C08996=1031.211,97.097,-98.859,168.789,43.801,158.206
C08997=1031.206,96.848,-98.839,168.786,43.803,158.206
C08998=1031.199,96.599,-98.821,168.784,43.804,158.206
C08999=1031.194,96.349,-98.802,168.781,43.806,158.206
C09000=1031.187,96.101,-98.782,168.779,43.808,158.206
C09001=1031.180,95.852,-98.764,168.776,43.809,158.206
C09002=1031.175,95.602,-98.744,168.775,43.811,158.206
C09003=1031.168,95.353,-98.726,168.772,43.812,158.206
C09004=1031.163,95.104,-98.706,168.769,43.814,158.207
C09005=1031.156,94.855,-98.688,168.768,43.816,158.207
C09006=1031.150,94.605,-98.669,168.765,43.818,158.207
C09007=1031.144,94.356,-98.650,168.762,43.819,158.207
C09008=1031.138,94.107,-98.631,168.760,43.821,158.207
C09009=1031.132,93.858,-98.612,168.758,43.823,158.207
C09010=1031.125,93.609,-98.593,168.755,43.824,158.207
C09011=1031.120,93.360,-98.573,168.753,43.826,158.207
C09012=1031.113,93.111,-98.555,168.751,43.827,158.208
C09013=1031.107,92.861,-98.535,168.748,43.829,158.208
C09014=1031.101,92.576,-98.514,168.746,43.831,158.208
C09015=1031.093,92.290,-98.492,168.743,43.833,158.208
C09016=1031.086,92.005,-98.470,168.741,43.835,158.208
C09017=1031.079,91.720,-98.449,168.737,43.836,158.208
C09018=1031.073,91.470,-98.431,168.735,43.838,158.208
C09019=1031.067,91.221,-98.411,168.733,43.840,158.208
C09020=1031.061,90.972,-98.393,168.730,43.842,158.209
C09021=1031.055,90.722,-98.373,168.728,43.843,158.209
C09022=1031.049,90.473,-98.355,168.726,43.845,158.209
C09023=1031.043,90.224,-98.336,168.723,43.847,158.209
C09024=1031.037,89.975,-98.317,168.721,43.848,158.209
C09025=1031.031,89.725,-98.298,168.718,43.850,158.209
C09026=1031.024,89.476,-98.279,168.716,43.851,158.209
C09027=1031.018,89.227,-98.260,168.713,43.853,158.209
C09028=1031.012,88.978,-98.242,168.712,43.855,158.210
C09029=1031.005,88.728,-98.224,168.709,43.856,158.210
C09030=1031.000,88.480,-98.206,168.706,43.858,158.210
C09031=1030.993,88.231,-98.187,168.704,43.860,158.210
C09032=1030.988,87.981,-98.168,168.702,43.862,158.210
C09033=1030.981,87.732,-98.149,168.699,43.864,158.210
C09034=1030.975,87.483,-98.130,168.697,43.865,158.210
C09035=1030.969,87.233,-98.112,168.695,43.866,158.210
C09036=1030.962,86.984,-98.094,168.692,43.868,158.210
C09037=1030.956,86.735,-98.075,168.690,43.870,158.211
C09038=1030.949,86.486,-98.056,168.687,43.872,158.211
C09039=1030.943,86.236,-98.038,168.686,43.874,158.211
C09040=1030.937,85.987,-98.019,168.683,43.876,158.211
C09041=1030.931,85.738,-98.001,168.680,43.877,158.211
C09042=1030.925,85.489,-97.982,168.678,43.879,158.211
C09043=1030.919,85.240,-97.964,168.676,43.881,158.211
C09044=1030.913,84.990,-97.946,168.673,43.882,158.211
C09045=1030.906,84.741,-97.927,168.671,43.884,158.212
C09046=1030.900,84.492,-97.908,168.669,43.885,158.212
C09047=1030.894,84.242,-97.890,168.666,43.887,158.212
C09048=1030.888,83.993,-97.871,168.664,43.889,158.212
C09049=1030.882,83.744,-97.853,168.661,43.891,158.212
C09050=1030.876,83.495,-97.834,168.659,43.892,158.212
C09051=1030.870,83.246,-97.816,168.657,43.894,158.212
C09052=1030.863,82.997,-97.798,168.654,43.896,158.212
C09053=1030.857,82.747,-97.779,168.653,43.898,158.213
C09054=1030.851,82.498,-97.761,168.650,43.899,158.213
C09055=1030.844,82.249,-97.743,168.647,43.901,158.213
C09056=1030.839,81.999,-97.723,168.646,43.902,158.213
C09057=1030.833,81.750,-97.706,168.643,43.904,158.213
C09058=1030.827,81.501,-97.687,168.640,43.906,158.213
C09059=1030.820,81.252,-97.668,168.637,43.907,158.213
C09060=1030.814,81.002,-97.650,168.636,43.909,158.213
C09061=1030.808,80.753,-97.632,168.633,43.911,158.213
C09062=1030.802,80.505,-97.614,168.631,43.913,158.214
C09063=1030.796,80.255,-97.596,168.629,43.914,158.214
C09064=1030.789,80.006,-97.577,168.626,43.916,158.214
C09065=1030.784,79.756,-97.558,168.624,43.918,158.214
C09066=1030.777,79.506,-97.540,168.622,43.919,158.214
C09067=1030.772,79.258,-97.522,168.619,43.921,158.214
C09068=1030.766,79.008,-97.504,168.617,43.923,158.214
C09069=1030.759,78.759,-97.485,168.615,43.924,158.214
C09070=1030.753,78.509,-97.467,168.612,43.926,158.215
C09071=1030.747,78.261,-97.449,168.610,43.927,158.215
C09072=1030.741,78.011,-97.431,168.608,43.929,158.215
C09073=1030.735,77.762,-97.412,168.605,43.931,158.215
C09074=1030.728,77.512,-97.394,168.603,43.933,158.215
C09075=1030.722,77.263,-97.376,168.600,43.934,158.215
C09076=1030.717,77.014,-97.358,168.598,43.936,158.215
C09077=1030.710,76.765,-97.339,168.596,43.938,158.215
C09078=1030.703,76.480,-97.319,168.593,43.940,158.215
C09079=1030.696,76.195,-97.298,168.591,43.941,158.216
C09080=1030.689,75.908,-97.277,168.588,43.943,158.216
C09081=1030.682,75.623,-97.257,168.585,43.946,158.216
C09082=1030.676,75.374,-97.238,168.583,43.947,158.216
C09083=1030.669,75.124,-97.221,168.580,43.949,158.216
C09084=1030.663,74.876,-97.203,168.578,43.951,158.216
C09085=1030.657,74.626,-97.185,168.576,43.953,158.216
C09086=1030.651,74.377,-97.167,168.573,43.955,158.217
C09087=1030.644,74.127,-97.148,168.571,43.956,158.217
C09088=1030.639,73.878,-97.130,168.568,43.958,158.217
C09089=1030.632,73.629,-97.113,168.566,43.959,158.217
C09090=1030.625,73.380,-97.094,168.564,43.961,158.217
C09091=1030.620,73.131,-97.077,168.561,43.963,158.217
C09092=1030.614,72.881,-97.059,168.560,43.965,158.217
C09093=1030.607,72.632,-97.040,168.557,43.967,158.218
C09094=1030.601,72.382,-97.022,168.554,43.968,158.218
C09095=1030.595,72.133,-97.005,168.552,43.970,158.218
C09096=1030.589,71.884,-96.987,168.550,43.972,158.218
C09097=1030.582,71.635,-96.969,168.547,43.973,158.218
C09098=1030.577,71.386,-96.951,168.545,43.975,158.218
C09099=1030.571,71.136,-96.933,168.543,43.976,158.218
C09100=1030.564,70.887,-96.915,168.540,43.978,158.218
C09101=1030.558,70.638,-96.898,168.538,43.980,158.218
C09102=1030.552,70.388,-96.880,168.536,43.982,158.219
C09103=1030.546,70.139,-96.861,168.534,43.984,158.219
C09104=1030.539,69.890,-96.844,168.531,43.985,158.219
C09105=1030.533,69.641,-96.826,168.528,43.987,158.219
C09106=1030.527,69.391,-96.808,168.526,43.989,158.219
C09107=1030.522,69.142,-96.791,168.524,43.991,158.219
C09108=1030.515,68.893,-96.772,168.521,43.992,158.219
C09109=1030.508,68.643,-96.755,168.520,43.994,158.219
C09110=1030.503,68.394,-96.737,168.517,43.995,158.219
C09111=1030.496,68.145,-96.720,168.514,43.997,158.220
C09112=1030.490,67.895,-96.702,168.512,43.999,158.220
C09113=1030.484,67.646,-96.684,168.510,44.001,158.220
C09114=1030.477,67.397,-96.666,168.507,44.003,158.220
C09115=1030.471,67.147,-96.648,168.505,44.005,158.220
C09116=1030.466,66.898,-96.631,168.503,44.006,158.220
C09117=1030.459,66.649,-96.613,168.500,44.008,158.220
C09118=1030.453,66.399,-96.595,168.498,44.010,158.221
C09119=1030.447,66.150,-96.578,168.495,44.011,158.221
C09120=1030.440,65.901,-96.561,168.494,44.013,158.221
C09121=1030.435,65.652,-96.543,168.491,44.015,158.221
C09122=1030.428,65.402,-96.526,168.488,44.017,158.221
C09123=1030.422,65.153,-96.508,168.487,44.019,158.221
C09124=1030.416,64.904,-96.490,168.484,44.020,158.221
C09125=1030.409,64.654,-96.473,168.481,44.022,158.221
C09126=1030.403,64.406,-96.455,168.479,44.024,158.222
C09127=1030.397,64.156,-96.437,168.477,44.025,158.222
C09128=1030.390,63.907,-96.419,168.475,44.027,158.222
C09129=1030.384,63.658,-96.402,168.472,44.029,158.222
C09130=1030.378,63.408,-96.384,168.469,44.030,158.222
C09131=1030.372,63.159,-96.368,168.468,44.032,158.222
C09132=1030.366,62.909,-96.350,168.465,44.034,158.222
C09133=1030.359,62.660,-96.333,168.463,44.037,158.223
C09134=1030.353,62.411,-96.316,168.460,44.039,158.223
C09135=1030.346,62.161,-96.299,168.458,44.040,158.223
C09136=1030.341,61.912,-96.281,168.456,44.042,158.223
C09137=1030.334,61.663,-96.264,168.453,44.043,158.223
C09138=1030.327,61.413,-96.246,168.450,44.045,158.223
C09139=1030.321,61.164,-96.229,168.449,44.047,158.223
C09140=1030.315,60.914,-96.212,168.446,44.049,158.223
C09141=1030.308,60.666,-96.195,168.444,44.051,158.224
C09142=1030.302,60.380,-96.175,168.441,44.053,158.224
C09143=1030.294,60.095,-96.155,168.439,44.055,158.224
C09144=1030.287,59.809,-96.135,168.435,44.057,158.224
C09145=1030.280,59.523,-96.115,168.432,44.059,158.224
C09146=1030.273,59.274,-96.098,168.431,44.061,158.224
C09147=1030.267,59.024,-96.082,168.428,44.063,158.224
C09148=1030.260,58.775,-96.064,168.426,44.065,158.225
C09149=1030.254,58.526,-96.047,168.423,44.067,158.225
C09150=1030.248,58.276,-96.029,168.421,44.068,158.225
C09151=1030.241,58.027,-96.012,168.419,44.070,158.225
C09152=1030.235,57.777,-95.995,168.416,44.072,158.225
C09153=1030.229,57.528,-95.978,168.414,44.074,158.225
C09154=1030.222,57.279,-95.961,168.412,44.076,158.226
C09155=1030.216,57.030,-95.944,168.409,44.078,158.226
C09156=1030.210,56.780,-95.927,168.407,44.080,158.226
C09157=1030.204,56.531,-95.910,168.404,44.082,158.226
C09158=1030.197,56.282,-95.892,168.402,44.084,158.226
C09159=1030.191,56.033,-95.875,168.400,44.085,158.226
C09160=1030.185,55.783,-95.858,168.397,44.087,158.226
C09161=1030.179,55.534,-95.841,168.395,44.088,158.226
C09162=1030.172,55.284,-95.824,168.393,44.090,158.227
C09163=1030.167,55.035,-95.807,168.390,44.092,158.227
C09164=1030.160,54.785,-95.790,168.388,44.094,158.227
C09165=1030.154,54.537,-95.773,168.385,44.096,158.227
C09166=1030.147,54.287,-95.756,168.384,44.098,158.227
C09167=1030.142,54.038,-95.739,168.381,44.100,158.227
C09168=1030.135,53.789,-95.722,168.378,44.101,158.227
C09169=1030.129,53.539,-95.705,168.376,44.103,158.227
C09170=1030.123,53.290,-95.688,168.374,44.105,158.228
C09171=1030.116,53.040,-95.670,168.371,44.106,158.228
C09172=1030.110,52.791,-95.654,168.369,44.108,158.228
C09173=1030.104,52.542,-95.636,168.366,44.110,158.228
C09174=1030.097,52.293,-95.619,168.365,44.112,158.228
C09175=1030.092,52.043,-95.603,168.362,44.114,158.228
C09176=1030.085,51.794,-95.585,168.359,44.116,158.228
C09177=1030.079,51.544,-95.569,168.357,44.118,158.228
C09178=1030.072,51.295,-95.552,168.355,44.119,158.229
C09179=1030.067,51.046,-95.534,168.352,44.121,158.229
C09180=1030.060,50.796,-95.517,168.350,44.122,158.229
C09181=1030.054,50.547,-95.501,168.347,44.124,158.229
C09182=1030.048,50.298,-95.484,168.346,44.126,158.229
C09183=1030.042,50.048,-95.466,168.343,44.128,158.229
C09184=1030.036,49.799,-95.450,168.340,44.130,158.229
C09185=1030.030,49.550,-95.433,168.339,44.131,158.229
C09186=1030.023,49.300,-95.416,168.336,44.133,158.230
C09187=1030.018,49.051,-95.399,168.333,44.135,158.230
C09188=1030.011,48.801,-95.382,168.331,44.137,158.230
C09189=1030.005,48.552,-95.365,168.329,44.138,158.230
C09190=1029.999,48.303,-95.349,168.326,44.140,158.230
C09191=1029.993,48.053,-95.331,168.324,44.142,158.230
C09192=1029.987,47.804,-95.315,168.322,44.143,158.230
C09193=1029.981,47.555,-95.298,168.320,44.145,158.230
C09194=1029.974,47.305,-95.281,168.317,44.147,158.230
C09195=1029.969,47.056,-95.264,168.314,44.149,158.231
C09196=1029.963,46.806,-95.247,168.313,44.150,158.231
C09197=1029.956,46.557,-95.230,168.310,44.152,158.231
C09198=1029.950,46.308,-95.214,168.307,44.154,158.231
C09199=1029.944,46.059,-95.196,168.305,44.156,158.231
C09200=1029.938,45.809,-95.180,168.303,44.157,158.231
C09201=1029.932,45.560,-95.163,168.300,44.159,158.231
C09202=1029.926,45.311,-95.146,168.298,44.161,158.231
C09203=1029.919,45.062,-95.129,168.296,44.162,158.232
C09204=1029.913,44.811,-95.112,168.294,44.164,158.232
C09205=1029.908,44.562,-95.096,168.291,44.166,158.232
C09206=1029.900,44.276,-95.077,168.288,44.168,158.232
C09207=1029.894,43.991,-95.058,168.286,44.169,158.232
C09208=1029.887,43.705,-95.038,168.283,44.171,158.232
C09209=1029.879,43.418,-95.019,168.280,44.173,158.232
C09210=1029.873,43.170,-95.002,168.278,44.175,158.232
C09211=1029.868,42.920,-94.985,168.275,44.177,158.232
C09212=1029.861,42.670,-94.969,168.274,44.179,158.233
C09213=1029.855,42.421,-94.953,168.271,44.181,158.233
C09214=1029.848,42.172,-94.936,168.268,44.183,158.233
C09215=1029.843,41.923,-94.920,168.266,44.185,158.233
C09216=1029.836,41.673,-94.903,168.264,44.186,158.233
C09217=1029.830,41.423,-94.887,168.261,44.188,158.233
C09218=1029.824,41.175,-94.870,168.259,44.189,158.233
C09219=1029.817,40.925,-94.853,168.256,44.191,158.233
C09220=1029.811,40.675,-94.837,168.254,44.193,158.233
C09221=1029.805,40.426,-94.821,168.252,44.195,158.234
C09222=1029.799,40.177,-94.804,168.249,44.197,158.234
C09223=1029.792,39.927,-94.787,168.247,44.199,158.234
C09224=1029.787,39.678,-94.771,168.244,44.200,158.234
C09225=1029.781,39.429,-94.755,168.242,44.202,158.234
C09226=1029.775,39.179,-94.738,168.240,44.204,158.234
C09227=1029.768,38.930,-94.722,168.237,44.206,158.234
C09228=1029.762,38.680,-94.705,168.235,44.208,158.234
C09229=1029.756,38.431,-94.689,168.233,44.209,158.235
C09230=1029.750,38.182,-94.672,168.230,44.211,158.235
C09231=1029.743,37.933,-94.657,168.228,44.212,158.235
C09232=1029.737,37.683,-94.640,168.225,44.214,158.235
C09233=1029.731,37.433,-94.624,168.223,44.216,158.235
C09234=1029.725,37.184,-94.608,168.221,44.218,158.235
C09235=1029.719,36.935,-94.591,168.218,44.220,158.235
C09236=1029.713,36.686,-94.574,168.216,44.222,158.235
C09237=1029.706,36.436,-94.558,168.213,44.224,158.236
C09238=1029.699,36.187,-94.542,168.211,44.226,158.236
C09239=1029.693,35.937,-94.526,168.209,44.227,158.236
C09240=1029.687,35.688,-94.510,168.206,44.229,158.236
C09241=1029.681,35.439,-94.494,168.204,44.231,158.236
C09242=1029.674,35.189,-94.477,168.201,44.233,158.236
C09243=1029.668,34.940,-94.461,168.199,44.235,158.236
C09244=1029.662,34.690,-94.445,168.197,44.237,158.237
C09245=1029.656,34.441,-94.429,168.194,44.239,158.237
C09246=1029.650,34.192,-94.413,168.192,44.241,158.237
C09247=1029.644,33.943,-94.397,168.189,44.242,158.237
C09248=1029.637,33.692,-94.381,168.187,44.244,158.237
C09249=1029.631,33.443,-94.365,168.185,44.246,158.237
C09250=1029.625,33.193,-94.349,168.182,44.248,158.237
C09251=1029.618,32.944,-94.333,168.179,44.249,158.237
C09252=1029.612,32.695,-94.317,168.177,44.251,158.237
C09253=1029.606,32.446,-94.301,168.175,44.253,158.238
C09254=1029.600,32.196,-94.284,168.173,44.255,158.238
C09255=1029.593,31.947,-94.268,168.170,44.257,158.238
C09256=1029.587,31.697,-94.252,168.167,44.259,158.238
C09257=1029.581,31.448,-94.236,168.165,44.261,158.238
C09258=1029.574,31.199,-94.220,168.163,44.263,158.238
C09259=1029.568,30.950,-94.204,168.161,44.265,158.238
C09260=1029.563,30.700,-94.188,168.158,44.266,158.238
C09261=1029.556,30.451,-94.173,168.155,44.268,158.239
C09262=1029.550,30.201,-94.156,168.153,44.270,158.239
C09263=1029.544,29.951,-94.140,168.151,44.271,158.239
C09264=1029.537,29.702,-94.124,168.148,44.273,158.239
C09265=1029.531,29.453,-94.108,168.146,44.275,158.239
C09266=1029.525,29.203,-94.092,168.143,44.277,158.239
C09267=1029.519,28.954,-94.077,168.142,44.279,158.239
C09268=1029.513,28.704,-94.060,168.139,44.281,158.239
C09269=1029.507,28.455,-94.044,168.136,44.282,158.239
C09270=1029.499,28.169,-94.026,168.134,44.285,158.240
C09271=1029.493,27.883,-94.007,168.131,44.287,158.240
C09272=1029.485,27.597,-93.990,168.128,44.289,158.240
C09273=1029.478,27.311,-93.972,168.125,44.291,158.240
C09274=1029.472,27.062,-93.955,168.122,44.293,158.240
C09275=1029.466,26.812,-93.940,168.120,44.294,158.240
C09276=1029.460,26.563,-93.924,168.118,44.296,158.240
C09277=1029.453,26.314,-93.909,168.116,44.298,158.241
C09278=1029.447,26.065,-93.892,168.113,44.300,158.241
C09279=1029.441,25.815,-93.877,168.111,44.302,158.241
C09280=1029.435,25.565,-93.861,168.108,44.304,158.241
C09281=1029.428,25.316,-93.846,168.105,44.306,158.241
C09282=1029.422,25.067,-93.830,168.104,44.308,158.241
C09283=1029.416,24.817,-93.814,168.101,44.310,158.241
C09284=1029.409,24.567,-93.799,168.099,44.311,158.241
C09285=1029.403,24.318,-93.783,168.096,44.313,158.242
C09286=1029.396,24.069,-93.767,168.093,44.315,158.242
C09287=1029.390,23.819,-93.751,168.091,44.317,158.242
C09288=1029.384,23.570,-93.736,168.089,44.319,158.242
C09289=1029.378,23.320,-93.720,168.087,44.321,158.242
C09290=1029.371,23.071,-93.705,168.084,44.323,158.242
C09291=1029.365,22.822,-93.689,168.081,44.324,158.242
C09292=1029.359,22.572,-93.673,168.079,44.326,158.242
C09293=1029.352,22.323,-93.658,168.076,44.328,158.242
C09294=1029.347,22.073,-93.642,168.074,44.330,158.243
C09295=1029.340,21.824,-93.626,168.072,44.332,158.243
C09296=1029.334,21.574,-93.611,168.069,44.334,158.243
C09297=1029.328,21.325,-93.596,168.067,44.335,158.243
C09298=1029.322,21.076,-93.581,168.064,44.337,158.243
C09299=1029.316,20.826,-93.564,168.061,44.339,158.243
C09300=1029.310,20.577,-93.549,168.060,44.341,158.243
C09301=1029.304,20.327,-93.533,168.057,44.343,158.244
C09302=1029.297,20.078,-93.518,168.055,44.345,158.244
C09303=1029.291,19.828,-93.502,168.052,44.346,158.244
C09304=1029.285,19.579,-93.487,168.049,44.348,158.244
C09305=1029.278,19.330,-93.471,168.047,44.350,158.244
C09306=1029.273,19.080,-93.456,168.044,44.352,158.244
C09307=1029.266,18.831,-93.440,168.042,44.354,158.244
C09308=1029.259,18.581,-93.425,168.040,44.356,158.244
C09309=1029.253,18.332,-93.410,168.037,44.358,158.244
C09310=1029.247,18.082,-93.394,168.035,44.360,158.245
C09311=1029.241,17.832,-93.379,168.032,44.361,158.245
C09312=1029.234,17.583,-93.363,168.029,44.363,158.245
C09313=1029.228,17.333,-93.348,168.027,44.365,158.245
C09314=1029.222,17.084,-93.333,168.025,44.367,158.245
C09315=1029.216,16.835,-93.318,168.023,44.369,158.245
C09316=1029.210,16.586,-93.303,168.020,44.371,158.245
C09317=1029.204,16.336,-93.286,168.017,44.373,158.245
C09318=1029.197,16.087,-93.272,168.015,44.375,158.246
C09319=1029.191,15.837,-93.257,168.012,44.377,158.246
C09320=1029.184,15.588,-93.241,168.010,44.379,158.246
C09321=1029.178,15.338,-93.225,168.008,44.380,158.246
C09322=1029.172,15.088,-93.210,168.005,44.382,158.246
C09323=1029.165,14.839,-93.195,168.003,44.384,158.246
C09324=1029.160,14.590,-93.180,168.000,44.386,158.246
C09325=1029.154,14.340,-93.165,167.997,44.388,158.246
C09326=1029.148,14.091,-93.150,167.995,44.389,158.246
C09327=1029.141,13.842,-93.134,167.992,44.391,158.247
C09328=1029.135,13.592,-93.119,167.991,44.393,158.247
C09329=1029.129,13.342,-93.104,167.988,44.395,158.247
C09330=1029.122,13.092,-93.089,167.985,44.397,158.247
C09331=1029.116,12.843,-93.074,167.983,44.399,158.247
C09332=1029.110,12.594,-93.058,167.980,44.401,158.247
C09333=1029.104,12.345,-93.043,167.978,44.403,158.247
C09334=1029.095,12.060,-93.026,167.975,44.405,158.248
C09335=1029.089,11.775,-93.010,167.972,44.408,158.248
C09336=1029.082,11.490,-92.992,167.969,44.410,158.248
C09337=1029.074,11.206,-92.976,167.967,44.412,158.248
C09338=1029.068,10.956,-92.961,167.964,44.414,158.248
C09339=1029.061,10.707,-92.946,167.962,44.416,158.248
C09340=1029.055,10.457,-92.931,167.959,44.418,158.248
C09341=1029.049,10.208,-92.916,167.956,44.420,158.249
C09342=1029.043,9.959,-92.901,167.954,44.422,158.249
C09343=1029.036,9.709,-92.886,167.951,44.424,158.249
C09344=1029.030,9.460,-92.871,167.949,44.426,158.249
C09345=1029.023,9.210,-92.856,167.946,44.428,158.249
C09346=1029.017,8.960,-92.841,167.943,44.430,158.249
C09347=1029.011,8.711,-92.826,167.941,44.432,158.249
C09348=1029.005,8.462,-92.811,167.938,44.433,158.249
C09349=1028.998,8.212,-92.796,167.937,44.435,158.249
C09350=1028.992,7.963,-92.781,167.934,44.437,158.250
C09351=1028.986,7.714,-92.767,167.931,44.439,158.250
C09352=1028.980,7.464,-92.752,167.929,44.441,158.250
C09353=1028.973,7.214,-92.737,167.926,44.443,158.250
C09354=1028.967,6.965,-92.722,167.924,44.445,158.250
C09355=1028.961,6.715,-92.707,167.921,44.447,158.250
C09356=1028.955,6.466,-92.692,167.918,44.449,158.250
C09357=1028.949,6.216,-92.678,167.916,44.451,158.250
C09358=1028.942,5.967,-92.663,167.913,44.453,158.251
C09359=1028.936,5.718,-92.648,167.911,44.455,158.251
C09360=1028.930,5.468,-92.633,167.908,44.457,158.251
C09361=1028.924,5.218,-92.618,167.906,44.458,158.251
C09362=1028.917,4.969,-92.603,167.904,44.460,158.251
C09363=1028.911,4.720,-92.589,167.901,44.462,158.251
C09364=1028.905,4.470,-92.574,167.899,44.464,158.251
C09365=1028.899,4.220,-92.559,167.896,44.466,158.251
C09366=1028.893,3.971,-92.545,167.894,44.468,158.252
C09367=1028.887,3.721,-92.530,167.891,44.470,158.252
C09368=1028.880,3.472,-92.515,167.888,44.472,158.252
C09369=1028.874,3.222,-92.500,167.886,44.474,158.252
C09370=1028.868,2.973,-92.485,167.883,44.476,158.252
C09371=1028.862,2.723,-92.470,167.880,44.477,158.252
C09372=1028.856,2.474,-92.456,167.878,44.479,158.252
C09373=1028.849,2.225,-92.442,167.876,44.481,158.252
C09374=1028.843,1.975,-92.427,167.874,44.483,158.252
C09375=1028.837,1.725,-92.412,167.871,44.485,158.252
C09376=1028.831,1.476,-92.398,167.868,44.487,158.253
C09377=1028.824,1.226,-92.383,167.866,44.489,158.253
C09378=1028.819,0.978,-92.368,167.863,44.491,158.253
C09379=1028.812,0.728,-92.353,167.861,44.493,158.253
C09380=1028.806,0.478,-92.339,167.858,44.494,158.253
C09381=1028.800,0.229,-92.325,167.855,44.496,158.253
C09382=1028.794,-0.021,-92.310,167.853,44.498,158.253
C09383=1028.788,-0.271,-92.295,167.850,44.500,158.253
C09384=1028.782,-0.520,-92.280,167.847,44.502,158.253
C09385=1028.776,-0.770,-92.266,167.846,44.503,158.254
C09386=1028.770,-1.019,-92.251,167.843,44.505,158.254
C09387=1028.764,-1.269,-92.236,167.841,44.507,158.254
C09388=1028.757,-1.518,-92.221,167.838,44.509,158.254
C09389=1028.752,-1.768,-92.207,167.835,44.511,158.254
C09390=1028.745,-2.017,-92.193,167.833,44.513,158.254
C09391=1028.739,-2.266,-92.179,167.830,44.514,158.254
C09392=1028.732,-2.516,-92.164,167.827,44.516,158.254
C09393=1028.727,-2.765,-92.150,167.825,44.518,158.254
C09394=1028.721,-3.015,-92.135,167.822,44.520,158.254
C09395=1028.714,-3.265,-92.120,167.820,44.522,158.255
C09396=1028.709,-3.514,-92.106,167.817,44.524,158.255
C09397=1028.702,-3.764,-92.091,167.815,44.526,158.255
C09398=1028.695,-4.071,-92.073,167.812,44.528,158.255
C09399=1028.687,-4.380,-92.056,167.808,44.531,158.255
C09400=1028.679,-4.688,-92.038,167.805,44.533,158.255
C09401=1028.671,-4.996,-92.021,167.802,44.536,158.255
C09402=1028.665,-5.246,-92.006,167.800,44.538,158.255
C09403=1028.658,-5.495,-91.992,167.797,44.539,158.256
C09404=1028.653,-5.745,-91.978,167.795,44.541,158.256
C09405=1028.646,-5.994,-91.963,167.792,44.543,158.256
C09406=1028.640,-6.232,-91.951,167.789,44.545,158.256
C09407=1028.634,-6.468,-91.937,167.787,44.547,158.256
C09408=1028.629,-6.705,-91.923,167.784,44.549,158.256
C09409=1028.622,-6.942,-91.910,167.782,44.551,158.256
C09410=1028.616,-7.178,-91.897,167.779,44.553,158.256
C09411=1028.611,-7.415,-91.883,167.778,44.555,158.257
C09412=1028.605,-7.652,-91.870,167.775,44.557,158.257
C09413=1028.599,-7.889,-91.856,167.772,44.558,158.257
C09414=1028.593,-8.138,-91.842,167.770,44.560,158.257
C09415=1028.587,-8.388,-91.828,167.767,44.563,158.257
C09416=1028.580,-8.637,-91.814,167.765,44.565,158.257
C09417=1028.574,-8.887,-91.800,167.762,44.567,158.257
C09418=1028.568,-9.136,-91.786,167.759,44.569,158.257
C09419=1028.562,-9.386,-91.772,167.757,44.571,158.257
C09420=1028.556,-9.636,-91.758,167.754,44.572,158.258
C09421=1028.549,-9.885,-91.743,167.752,44.574,158.258
C09422=1028.543,-10.134,-91.730,167.749,44.576,158.258
C09423=1028.537,-10.384,-91.716,167.746,44.578,158.258
C09424=1028.531,-10.633,-91.701,167.744,44.580,158.258
C09425=1028.524,-10.883,-91.688,167.741,44.582,158.258
C09426=1028.518,-11.132,-91.673,167.739,44.584,158.258
C09427=1028.511,-11.382,-91.660,167.736,44.586,158.258
C09428=1028.506,-11.632,-91.646,167.733,44.588,158.258
C09429=1028.500,-11.881,-91.631,167.731,44.590,158.259
C09430=1028.493,-12.131,-91.617,167.728,44.591,158.259
C09431=1028.488,-12.380,-91.604,167.725,44.593,158.259
C09432=1028.481,-12.630,-91.589,167.723,44.595,158.259
C09433=1028.475,-12.879,-91.575,167.720,44.597,158.259
C09434=1028.468,-13.129,-91.562,167.718,44.599,158.259
C09435=1028.463,-13.379,-91.548,167.715,44.601,158.259
C09436=1028.456,-13.627,-91.534,167.712,44.603,158.259
C09437=1028.450,-13.878,-91.520,167.710,44.605,158.259
C09438=1028.445,-14.127,-91.506,167.707,44.607,158.259
C09439=1028.438,-14.376,-91.492,167.705,44.609,158.260
C09440=1028.432,-14.626,-91.478,167.702,44.611,158.260
C09441=1028.426,-14.876,-91.464,167.699,44.613,158.260
C09442=1028.420,-15.126,-91.450,167.697,44.615,158.260
C09443=1028.414,-15.375,-91.437,167.694,44.617,158.260
C09444=1028.408,-15.624,-91.422,167.692,44.619,158.260
C09445=1028.401,-15.874,-91.409,167.689,44.621,158.260
C09446=1028.395,-16.123,-91.395,167.687,44.623,158.260
C09447=1028.389,-16.374,-91.381,167.684,44.625,158.260
C09448=1028.383,-16.623,-91.368,167.681,44.627,158.261
C09449=1028.376,-16.872,-91.355,167.678,44.629,158.261
C09450=1028.370,-17.122,-91.340,167.675,44.631,158.261
C09451=1028.364,-17.372,-91.327,167.673,44.633,158.261
C09452=1028.358,-17.621,-91.314,167.670,44.635,158.261
C09453=1028.351,-17.870,-91.299,167.668,44.637,158.261
C09454=1028.345,-18.120,-91.286,167.665,44.639,158.261
C09455=1028.339,-18.369,-91.272,167.662,44.641,158.261
C09456=1028.332,-18.619,-91.259,167.660,44.643,158.261
C09457=1028.327,-18.869,-91.245,167.657,44.645,158.262
C09458=1028.321,-19.118,-91.232,167.655,44.647,158.262
C09459=1028.314,-19.368,-91.218,167.652,44.649,158.262
C09460=1028.308,-19.617,-91.205,167.649,44.651,158.262
C09461=1028.302,-19.867,-91.191,167.647,44.653,158.262
C09462=1028.295,-20.147,-91.176,167.643,44.656,158.262
C09463=1028.288,-20.429,-91.161,167.641,44.658,158.262
C09464=1028.281,-20.710,-91.145,167.637,44.660,158.262
C09465=1028.273,-20.991,-91.130,167.635,44.662,158.262
C09466=1028.268,-21.241,-91.117,167.632,44.665,158.263
C09467=1028.262,-21.491,-91.103,167.630,44.667,158.263
C09468=1028.255,-21.740,-91.090,167.627,44.669,158.263
C09469=1028.249,-21.990,-91.076,167.623,44.671,158.263
C09470=1028.243,-22.239,-91.063,167.621,44.673,158.263
C09471=1028.237,-22.489,-91.049,167.618,44.675,158.263
C09472=1028.230,-22.739,-91.036,167.616,44.677,158.263
C09473=1028.224,-22.988,-91.022,167.613,44.679,158.263
C09474=1028.219,-23.237,-91.008,167.611,44.680,158.264
C09475=1028.212,-23.487,-90.995,167.608,44.682,158.264
C09476=1028.206,-23.737,-90.982,167.605,44.684,158.264
C09477=1028.199,-23.986,-90.968,167.603,44.686,158.264
C09478=1028.194,-24.235,-90.954,167.600,44.688,158.264
C09479=1028.188,-24.485,-90.942,167.598,44.690,158.264
C09480=1028.182,-24.735,-90.929,167.595,44.692,158.264
C09481=1028.175,-24.985,-90.915,167.592,44.694,158.264
C09482=1028.170,-25.234,-90.901,167.590,44.696,158.264
C09483=1028.163,-25.483,-90.888,167.586,44.698,158.264
C09484=1028.157,-25.733,-90.875,167.584,44.700,158.265
C09485=1028.151,-25.983,-90.862,167.581,44.702,158.265
C09486=1028.146,-26.232,-90.848,167.578,44.704,158.265
C09487=1028.139,-26.482,-90.835,167.576,44.706,158.265
C09488=1028.133,-26.731,-90.821,167.573,44.708,158.265
C09489=1028.126,-26.981,-90.808,167.571,44.710,158.265
C09490=1028.121,-27.231,-90.795,167.568,44.712,158.265
C09491=1028.115,-27.480,-90.782,167.565,44.714,158.265
C09492=1028.108,-27.730,-90.768,167.563,44.716,158.265
C09493=1028.102,-27.979,-90.755,167.560,44.718,158.265
C09494=1028.096,-28.229,-90.742,167.557,44.720,158.266
C09495=1028.090,-28.478,-90.729,167.554,44.722,158.266
C09496=1028.084,-28.728,-90.716,167.552,44.725,158.266
C09497=1028.078,-28.978,-90.703,167.549,44.727,158.266
C09498=1028.072,-29.227,-90.690,167.547,44.729,158.266
C09499=1028.064,-29.477,-90.677,167.544,44.731,158.266
C09500=1028.058,-29.726,-90.664,167.541,44.733,158.266
C09501=1028.052,-29.976,-90.651,167.538,44.735,158.266
C09502=1028.046,-30.226,-90.638,167.535,44.737,158.266
C09503=1028.040,-30.475,-90.625,167.533,44.739,158.267
C09504=1028.034,-30.724,-90.612,167.530,44.741,158.267
C09505=1028.028,-30.974,-90.599,167.528,44.743,158.267
C09506=1028.021,-31.223,-90.586,167.525,44.745,158.267
C09507=1028.015,-31.474,-90.573,167.521,44.748,158.267
C09508=1028.009,-31.723,-90.560,167.519,44.750,158.267
C09509=1028.003,-31.973,-90.547,167.516,44.752,158.267
C09510=1027.997,-32.222,-90.534,167.514,44.754,158.267
C09511=1027.991,-32.472,-90.521,167.511,44.755,158.267
C09512=1027.985,-32.721,-90.508,167.508,44.757,158.268
C09513=1027.978,-32.971,-90.495,167.506,44.759,158.268
C09514=1027.972,-33.221,-90.482,167.502,44.762,158.268
C09515=1027.966,-33.470,-90.469,167.500,44.764,158.268
C09516=1027.960,-33.720,-90.457,167.497,44.766,158.268
C09517=1027.954,-33.969,-90.443,167.495,44.768,158.268
C09518=1027.948,-34.219,-90.431,167.492,44.770,158.268
C09519=1027.942,-34.468,-90.417,167.490,44.772,158.268
C09520=1027.936,-34.718,-90.405,167.487,44.774,158.268
C09521=1027.930,-34.968,-90.392,167.483,44.776,158.269
C09522=1027.924,-35.217,-90.379,167.481,44.778,158.269
C09523=1027.917,-35.467,-90.367,167.478,44.780,158.269
C09524=1027.911,-35.716,-90.354,167.476,44.782,158.269
C09525=1027.905,-35.966,-90.341,167.473,44.784,158.269
C09526=1027.898,-36.246,-90.326,167.470,44.787,158.269
C09527=1027.891,-36.527,-90.312,167.467,44.789,158.269
C09528=1027.884,-36.807,-90.298,167.463,44.791,158.269
C09529=1027.877,-37.087,-90.284,167.461,44.794,158.270
C09530=1027.871,-37.337,-90.270,167.458,44.796,158.270
C09531=1027.865,-37.587,-90.258,167.455,44.798,158.270
C09532=1027.859,-37.836,-90.244,167.452,44.800,158.270
C09533=1027.853,-38.086,-90.232,167.450,44.802,158.270
C09534=1027.847,-38.336,-90.219,167.447,44.804,158.270
C09535=1027.842,-38.584,-90.206,167.444,44.806,158.270
C09536=1027.836,-38.834,-90.194,167.442,44.808,158.270
C09537=1027.830,-39.084,-90.181,167.438,44.810,158.270
C09538=1027.823,-39.333,-90.169,167.436,44.812,158.270
C09539=1027.817,-39.583,-90.156,167.433,44.814,158.270
C09540=1027.811,-39.833,-90.144,167.431,44.817,158.271
C09541=1027.804,-40.082,-90.132,167.428,44.819,158.271
C09542=1027.799,-40.332,-90.119,167.424,44.821,158.271
C09543=1027.792,-40.581,-90.106,167.422,44.823,158.271
C09544=1027.786,-40.831,-90.094,167.419,44.825,158.271
C09545=1027.780,-41.081,-90.081,167.417,44.827,158.271
C09546=1027.774,-41.331,-90.069,167.413,44.830,158.271
C09547=1027.767,-41.580,-90.057,167.411,44.832,158.271
C09548=1027.761,-41.830,-90.044,167.408,44.834,158.271
C09549=1027.755,-42.079,-90.031,167.406,44.836,158.272
C09550=1027.748,-42.329,-90.019,167.403,44.838,158.272
C09551=1027.743,-42.578,-90.007,167.400,44.840,158.272
C09552=1027.737,-42.828,-89.994,167.397,44.842,158.272
C09553=1027.731,-43.078,-89.982,167.394,44.844,158.272
C09554=1027.725,-43.327,-89.970,167.392,44.846,158.272
C09555=1027.719,-43.577,-89.957,167.389,44.848,158.272
C09556=1027.712,-43.826,-89.945,167.386,44.851,158.272
C09557=1027.706,-44.076,-89.932,167.383,44.853,158.273
C09558=1027.700,-44.326,-89.919,167.381,44.855,158.273
C09559=1027.694,-44.575,-89.908,167.378,44.857,158.273
C09560=1027.688,-44.825,-89.895,167.375,44.859,158.273
C09561=1027.682,-45.075,-89.883,167.372,44.861,158.273
C09562=1027.676,-45.324,-89.871,167.369,44.863,158.273
C09563=1027.670,-45.574,-89.858,167.367,44.865,158.273
C09564=1027.664,-45.824,-89.846,167.364,44.868,158.273
C09565=1027.658,-46.073,-89.834,167.361,44.870,158.273
C09566=1027.652,-46.323,-89.821,167.358,44.872,158.273
C09567=1027.646,-46.573,-89.809,167.356,44.874,158.274
C09568=1027.639,-46.822,-89.797,167.353,44.876,158.274
C09569=1027.633,-47.072,-89.784,167.349,44.878,158.274
C09570=1027.627,-47.321,-89.773,167.347,44.880,158.274
C09571=1027.621,-47.571,-89.760,167.344,44.882,158.274
C09572=1027.615,-47.821,-89.748,167.342,44.885,158.274
C09573=1027.609,-48.070,-89.736,167.339,44.887,158.274
C09574=1027.603,-48.320,-89.724,167.336,44.889,158.274
C09575=1027.598,-48.569,-89.711,167.333,44.891,158.274
C09576=1027.591,-48.819,-89.699,167.330,44.893,158.274
C09577=1027.585,-49.069,-89.686,167.328,44.895,158.275
C09578=1027.579,-49.318,-89.675,167.324,44.897,158.275
C09579=1027.573,-49.568,-89.662,167.322,44.899,158.275
C09580=1027.567,-49.818,-89.650,167.319,44.902,158.275
C09581=1027.561,-50.067,-89.638,167.317,44.904,158.275
C09582=1027.556,-50.317,-89.626,167.313,44.906,158.275
C09583=1027.550,-50.567,-89.614,167.311,44.908,158.275
C09584=1027.543,-50.816,-89.602,167.308,44.910,158.275
C09585=1027.536,-51.066,-89.590,167.305,44.912,158.275
C09586=1027.530,-51.316,-89.577,167.302,44.915,158.276
C09587=1027.525,-51.565,-89.566,167.299,44.917,158.276
C09588=1027.518,-51.815,-89.555,167.297,44.919,158.276
C09589=1027.511,-52.064,-89.543,167.293,44.922,158.276
C09590=1027.505,-52.346,-89.529,167.291,44.924,158.276
C09591=1027.498,-52.625,-89.516,167.287,44.927,158.276
C09592=1027.491,-52.906,-89.503,167.284,44.930,158.276
C09593=1027.484,-53.187,-89.489,167.281,44.932,158.276
C09594=1027.478,-53.437,-89.478,167.278,44.934,158.277
C09595=1027.472,-53.686,-89.466,167.276,44.936,158.277
C09596=1027.466,-53.936,-89.454,167.272,44.939,158.277
C09597=1027.459,-54.186,-89.443,167.270,44.941,158.277
C09598=1027.453,-54.436,-89.431,167.267,44.943,158.277
C09599=1027.447,-54.685,-89.419,167.263,44.945,158.277
C09600=1027.440,-54.935,-89.408,167.261,44.948,158.277
C09601=1027.434,-55.185,-89.395,167.258,44.950,158.278
C09602=1027.428,-55.434,-89.384,167.255,44.952,158.278
C09603=1027.422,-55.684,-89.372,167.253,44.955,158.278
C09604=1027.416,-55.933,-89.361,167.250,44.957,158.278
C09605=1027.410,-56.183,-89.349,167.246,44.959,158.278
C09606=1027.404,-56.433,-89.337,167.244,44.962,158.278
C09607=1027.398,-56.682,-89.326,167.241,44.964,158.278
C09608=1027.391,-56.932,-89.314,167.238,44.966,158.278
C09609=1027.386,-57.182,-89.302,167.235,44.969,158.279
C09610=1027.380,-57.431,-89.291,167.233,44.971,158.279
C09611=1027.373,-57.681,-89.279,167.229,44.973,158.279
C09612=1027.367,-57.930,-89.268,167.227,44.975,158.279
C09613=1027.361,-58.180,-89.256,167.224,44.978,158.279
C09614=1027.355,-58.430,-89.244,167.221,44.980,158.279
C09615=1027.349,-58.679,-89.233,167.218,44.982,158.279
C09616=1027.343,-58.929,-89.221,167.216,44.984,158.279
C09617=1027.337,-59.178,-89.210,167.212,44.987,158.279
C09618=1027.330,-59.429,-89.198,167.210,44.989,158.279
C09619=1027.324,-59.678,-89.186,167.207,44.991,158.280
C09620=1027.319,-59.928,-89.175,167.204,44.994,158.280
C09621=1027.312,-60.178,-89.163,167.201,44.996,158.280
C09622=1027.306,-60.427,-89.152,167.198,44.998,158.280
C09623=1027.300,-60.677,-89.141,167.195,45.000,158.280
C09624=1027.295,-60.926,-89.129,167.192,45.002,158.280
C09625=1027.288,-61.177,-89.118,167.190,45.004,158.280
C09626=1027.282,-61.425,-89.106,167.186,45.007,158.280
C09627=1027.276,-61.676,-89.095,167.184,45.009,158.281
C09628=1027.270,-61.924,-89.083,167.181,45.011,158.281
C09629=1027.264,-62.175,-89.071,167.178,45.013,158.281
C09630=1027.259,-62.424,-89.060,167.175,45.016,158.281
C09631=1027.252,-62.674,-89.048,167.173,45.018,158.281
C09632=1027.246,-62.924,-89.038,167.169,45.020,158.281
C09633=1027.240,-63.174,-89.026,167.167,45.022,158.281
C09634=1027.235,-63.423,-89.014,167.164,45.025,158.281
C09635=1027.228,-63.673,-89.003,167.161,45.027,158.281
C09636=1027.222,-63.923,-88.992,167.158,45.029,158.282
C09637=1027.216,-64.172,-88.980,167.155,45.031,158.282
C09638=1027.210,-64.422,-88.969,167.152,45.034,158.282
C09639=1027.204,-64.672,-88.958,167.149,45.036,158.282
C09640=1027.198,-64.921,-88.946,167.147,45.038,158.282
C09641=1027.193,-65.171,-88.935,167.143,45.040,158.282
C09642=1027.186,-65.421,-88.924,167.141,45.043,158.282
C09643=1027.180,-65.670,-88.912,167.138,45.045,158.282
C09644=1027.174,-65.920,-88.901,167.135,45.047,158.282
C09645=1027.168,-66.169,-88.890,167.132,45.049,158.282
C09646=1027.163,-66.420,-88.878,167.130,45.052,158.283
C09647=1027.157,-66.669,-88.866,167.126,45.054,158.283
C09648=1027.151,-66.918,-88.856,167.124,45.056,158.283
C09649=1027.145,-67.168,-88.844,167.121,45.058,158.283
C09650=1027.139,-67.418,-88.833,167.118,45.061,158.283
C09651=1027.133,-67.667,-88.823,167.115,45.063,158.283
C09652=1027.127,-67.917,-88.810,167.112,45.065,158.283
C09653=1027.121,-68.167,-88.799,167.109,45.067,158.283
///RCONF 1,0,0,1,0,0,0,0,0,0,0,0,0,0,0,0,0,0,0,0,0,0,0,0
C09654=1027.114,-68.448,-88.787,167.107,45.070,158.283
C09655=1027.108,-68.731,-88.774,167.103,45.072,158.284
C09656=1027.101,-69.012,-88.761,167.100,45.075,158.284
C09657=1027.094,-69.294,-88.749,167.096,45.077,158.284
C09658=1027.088,-69.544,-88.738,167.094,45.080,158.284
C09659=1027.082,-69.794,-88.727,167.091,45.082,158.284
C09660=1027.077,-70.043,-88.715,167.087,45.084,158.284
C09661=1027.072,-70.293,-88.704,167.085,45.086,158.284
C09662=1027.065,-70.543,-88.693,167.082,45.088,158.284
C09663=1027.059,-70.792,-88.681,167.079,45.091,158.284
C09664=1027.053,-71.041,-88.671,167.076,45.093,158.285
C09665=1027.047,-71.292,-88.659,167.074,45.095,158.285
C09666=1027.041,-71.541,-88.648,167.070,45.097,158.285
C09667=1027.036,-71.791,-88.637,167.068,45.099,158.285
C09668=1027.030,-72.041,-88.626,167.065,45.102,158.285
C09669=1027.024,-72.291,-88.615,167.062,45.104,158.285
C09670=1027.019,-72.540,-88.604,167.059,45.106,158.285
C09671=1027.013,-72.790,-88.593,167.056,45.108,158.285
C09672=1027.006,-73.040,-88.582,167.053,45.110,158.285
C09673=1027.001,-73.289,-88.571,167.050,45.113,158.285
C09674=1026.995,-73.539,-88.560,167.048,45.115,158.286
C09675=1026.990,-73.789,-88.549,167.044,45.117,158.286
C09676=1026.984,-74.039,-88.537,167.042,45.119,158.286
C09677=1026.978,-74.288,-88.527,167.039,45.121,158.286
C09678=1026.972,-74.538,-88.516,167.036,45.124,158.286
C09679=1026.966,-74.787,-88.505,167.033,45.126,158.286
C09680=1026.959,-75.037,-88.494,167.030,45.129,158.286
C09681=1026.954,-75.287,-88.483,167.027,45.131,158.286
C09682=1026.948,-75.537,-88.473,167.025,45.133,158.286
C09683=1026.942,-75.786,-88.462,167.021,45.136,158.286
C09684=1026.936,-76.036,-88.451,167.019,45.138,158.287
C09685=1026.930,-76.286,-88.441,167.015,45.140,158.287
C09686=1026.924,-76.535,-88.430,167.013,45.143,158.287
C09687=1026.918,-76.785,-88.419,167.010,45.145,158.287
C09688=1026.913,-77.035,-88.409,167.007,45.148,158.287
C09689=1026.906,-77.285,-88.398,167.004,45.150,158.287
C09690=1026.901,-77.534,-88.387,167.001,45.152,158.287
C09691=1026.894,-77.784,-88.376,166.998,45.155,158.287
C09692=1026.888,-78.033,-88.365,166.995,45.157,158.287
C09693=1026.883,-78.283,-88.355,166.992,45.159,158.288
C09694=1026.877,-78.533,-88.344,166.990,45.162,158.288
C09695=1026.871,-78.783,-88.333,166.986,45.164,158.288
C09696=1026.865,-79.032,-88.322,166.983,45.166,158.288
C09697=1026.859,-79.282,-88.313,166.980,45.169,158.288
C09698=1026.853,-79.532,-88.302,166.977,45.171,158.288
C09699=1026.848,-79.781,-88.291,166.975,45.174,158.288
C09700=1026.842,-80.031,-88.281,166.972,45.176,158.288
C09701=1026.835,-80.281,-88.270,166.969,45.178,158.288
C09702=1026.829,-80.531,-88.259,166.966,45.181,158.289
C09703=1026.824,-80.781,-88.249,166.963,45.183,158.289
C09704=1026.817,-81.030,-88.239,166.960,45.186,158.289
C09705=1026.812,-81.280,-88.229,166.957,45.188,158.289
C09706=1026.805,-81.529,-88.218,166.954,45.191,158.289
C09707=1026.800,-81.779,-88.208,166.951,45.193,158.289
C09708=1026.793,-82.029,-88.198,166.948,45.196,158.289
C09709=1026.787,-82.279,-88.187,166.945,45.198,158.290
C09710=1026.782,-82.529,-88.177,166.942,45.200,158.290
C09711=1026.775,-82.778,-88.166,166.939,45.203,158.290
C09712=1026.770,-83.028,-88.156,166.936,45.205,158.290
C09713=1026.763,-83.277,-88.146,166.934,45.208,158.290
C09714=1026.758,-83.527,-88.136,166.930,45.210,158.290
C09715=1026.751,-83.777,-88.125,166.928,45.213,158.290
C09716=1026.746,-84.027,-88.115,166.924,45.215,158.290
C09717=1026.740,-84.276,-88.105,166.922,45.218,158.291
C09718=1026.733,-84.560,-88.093,166.918,45.221,158.291
C09719=1026.727,-84.844,-88.081,166.915,45.224,158.291
C09720=1026.719,-85.129,-88.070,166.911,45.226,158.291
C09721=1026.713,-85.412,-88.058,166.908,45.229,158.291
C09722=1026.707,-85.662,-88.048,166.906,45.232,158.291
C09723=1026.701,-85.912,-88.038,166.902,45.234,158.291
C09724=1026.695,-86.161,-88.028,166.900,45.237,158.292
C09725=1026.689,-86.411,-88.018,166.896,45.239,158.292
C09726=1026.684,-86.661,-88.007,166.894,45.242,158.292
C09727=1026.677,-86.910,-87.997,166.890,45.244,158.292
C09728=1026.672,-87.160,-87.986,166.888,45.246,158.292
C09729=1026.665,-87.410,-87.977,166.884,45.249,158.292
C09730=1026.660,-87.660,-87.967,166.882,45.251,158.292
C09731=1026.654,-87.909,-87.956,166.878,45.254,158.292
C09732=1026.648,-88.159,-87.946,166.876,45.256,158.293
C09733=1026.642,-88.409,-87.937,166.872,45.259,158.293
C09734=1026.636,-88.658,-87.926,166.870,45.261,158.293
C09735=1026.630,-88.908,-87.916,166.866,45.264,158.293
C09736=1026.625,-89.158,-87.906,166.864,45.266,158.293
C09737=1026.618,-89.408,-87.896,166.860,45.268,158.293
C09738=1026.613,-89.658,-87.886,166.858,45.271,158.293
C09739=1026.607,-89.907,-87.876,166.854,45.273,158.293
C09740=1026.601,-90.157,-87.865,166.852,45.276,158.294
C09741=1026.595,-90.407,-87.856,166.849,45.278,158.294
C09742=1026.589,-90.657,-87.845,166.846,45.281,158.294
C09743=1026.583,-90.907,-87.836,166.844,45.283,158.294
C09744=1026.577,-91.156,-87.825,166.840,45.286,158.294
C09745=1026.572,-91.405,-87.816,166.838,45.288,158.294
C09746=1026.566,-91.655,-87.806,166.834,45.290,158.294
C09747=1026.560,-91.905,-87.796,166.832,45.293,158.294
C09748=1026.554,-92.155,-87.785,166.828,45.295,158.294
C09749=1026.548,-92.404,-87.776,166.826,45.298,158.295
C09750=1026.543,-92.655,-87.765,166.822,45.300,158.295
C09751=1026.537,-92.904,-87.756,166.820,45.303,158.295
C09752=1026.531,-93.154,-87.746,166.816,45.305,158.295
C09753=1026.525,-93.403,-87.736,166.814,45.308,158.295
C09754=1026.520,-93.653,-87.726,166.810,45.310,158.295
C09755=1026.514,-93.903,-87.716,166.808,45.313,158.295
C09756=1026.508,-94.153,-87.706,166.804,45.315,158.295
C09757=1026.502,-94.403,-87.696,166.802,45.318,158.296
C09758=1026.497,-94.653,-87.686,166.798,45.320,158.296
C09759=1026.491,-94.902,-87.677,166.796,45.323,158.296
C09760=1026.485,-95.151,-87.666,166.792,45.325,158.296
C09761=1026.479,-95.401,-87.656,166.790,45.327,158.296
C09762=1026.474,-95.651,-87.646,166.787,45.330,158.296
C09763=1026.468,-95.901,-87.637,166.784,45.332,158.296
C09764=1026.463,-96.151,-87.627,166.782,45.335,158.296
C09765=1026.457,-96.400,-87.617,166.778,45.337,158.296
C09766=1026.451,-96.650,-87.607,166.776,45.340,158.297
C09767=1026.445,-96.900,-87.598,166.772,45.342,158.297
C09768=1026.439,-97.149,-87.588,166.770,45.345,158.297
C09769=1026.434,-97.399,-87.578,166.766,45.347,158.297
C09770=1026.428,-97.649,-87.569,166.764,45.349,158.297
C09771=1026.422,-97.899,-87.559,166.760,45.352,158.297
C09772=1026.417,-98.148,-87.549,166.758,45.354,158.297
C09773=1026.411,-98.398,-87.540,166.754,45.357,158.297
C09774=1026.404,-98.648,-87.530,166.752,45.359,158.298
C09775=1026.398,-98.898,-87.521,166.748,45.362,158.298
C09776=1026.393,-99.147,-87.511,166.745,45.365,158.298
C09777=1026.387,-99.397,-87.501,166.742,45.367,158.298
C09778=1026.381,-99.647,-87.492,166.739,45.370,158.298
C09779=1026.375,-99.897,-87.482,166.737,45.372,158.298
C09780=1026.370,-100.146,-87.474,166.733,45.375,158.298
C09781=1026.364,-100.396,-87.464,166.731,45.377,158.298
C09782=1026.357,-100.682,-87.452,166.727,45.380,158.299
C09783=1026.350,-100.968,-87.442,166.724,45.383,158.299
C09784=1026.344,-101.255,-87.431,166.721,45.387,158.299
C09785=1026.337,-101.541,-87.420,166.717,45.390,158.299
C09786=1026.331,-101.790,-87.411,166.714,45.392,158.299
C09787=1026.326,-102.040,-87.401,166.710,45.395,158.299
C09788=1026.320,-102.290,-87.391,166.708,45.397,158.299
C09789=1026.314,-102.540,-87.383,166.705,45.400,158.300
C09790=1026.308,-102.790,-87.373,166.702,45.403,158.300
C09791=1026.302,-103.040,-87.364,166.699,45.405,158.300
C09792=1026.297,-103.289,-87.354,166.696,45.408,158.300
C09793=1026.291,-103.539,-87.345,166.693,45.410,158.300
C09794=1026.285,-103.789,-87.336,166.690,45.413,158.300
C09795=1026.280,-104.038,-87.326,166.687,45.415,158.300
C09796=1026.274,-104.288,-87.317,166.684,45.417,158.300
C09797=1026.268,-104.539,-87.308,166.681,45.420,158.301
C09798=1026.263,-104.788,-87.298,166.679,45.423,158.301
C09799=1026.257,-105.038,-87.289,166.675,45.425,158.301
C09800=1026.251,-105.287,-87.280,166.672,45.428,158.301
C09801=1026.245,-105.537,-87.270,166.669,45.430,158.301
C09802=1026.239,-105.787,-87.261,166.666,45.433,158.301
C09803=1026.234,-106.037,-87.252,166.663,45.436,158.301
C09804=1026.228,-106.287,-87.243,166.660,45.438,158.301
C09805=1026.222,-106.536,-87.234,166.657,45.441,158.302
C09806=1026.217,-106.786,-87.224,166.654,45.444,158.302
C09807=1026.211,-107.035,-87.215,166.652,45.446,158.302
C09808=1026.205,-107.285,-87.205,166.648,45.449,158.302
C09809=1026.199,-107.536,-87.197,166.645,45.452,158.302
C09810=1026.194,-107.785,-87.187,166.642,45.454,158.302
C09811=1026.188,-108.035,-87.179,166.639,45.457,158.302
C09812=1026.182,-108.284,-87.169,166.637,45.460,158.303
C09813=1026.176,-108.535,-87.161,166.633,45.463,158.303
C09814=1026.171,-108.784,-87.151,166.631,45.465,158.303
C09815=1026.165,-109.034,-87.142,166.627,45.468,158.303
C09816=1026.159,-109.283,-87.133,166.624,45.471,158.303
C09817=1026.154,-109.534,-87.124,166.621,45.473,158.303
C09818=1026.148,-109.783,-87.115,166.618,45.476,158.303
C09819=1026.142,-110.033,-87.106,166.616,45.478,158.304
C09820=1026.137,-110.282,-87.097,166.612,45.481,158.304
C09821=1026.131,-110.533,-87.088,166.610,45.483,158.304
C09822=1026.124,-110.782,-87.080,166.606,45.486,158.304
C09823=1026.119,-111.032,-87.071,166.603,45.489,158.304
C09824=1026.113,-111.281,-87.062,166.601,45.492,158.304
C09825=1026.107,-111.531,-87.053,166.597,45.494,158.304
C09826=1026.102,-111.781,-87.044,166.595,45.497,158.305
C09827=1026.096,-112.031,-87.035,166.591,45.500,158.305
C09828=1026.090,-112.281,-87.026,166.589,45.502,158.305
C09829=1026.084,-112.530,-87.017,166.585,45.505,158.305
C09830=1026.079,-112.780,-87.008,166.582,45.508,158.305
///RCONF 1,0,0,0,0,0,0,0,0,0,0,0,0,0,0,0,0,0,0,0,0,0,0,0
C09831=1026.073,-113.031,-86.999,166.580,45.511,158.305
C09832=1026.067,-113.280,-86.990,166.576,45.513,158.305
C09833=1026.062,-113.529,-86.982,166.574,45.516,158.306
C09834=1026.056,-113.779,-86.972,166.570,45.518,158.306
C09835=1026.051,-114.029,-86.964,166.568,45.521,158.306
C09836=1026.045,-114.279,-86.955,166.565,45.523,158.306
C09837=1026.040,-114.529,-86.946,166.561,45.526,158.306
C09838=1026.033,-114.779,-86.937,166.559,45.529,158.306
C09839=1026.027,-115.028,-86.929,166.555,45.531,158.306
C09840=1026.022,-115.278,-86.920,166.553,45.534,158.307
C09841=1026.016,-115.528,-86.911,166.550,45.537,158.307
C09842=1026.011,-115.778,-86.902,166.546,45.540,158.307
C09843=1026.005,-116.028,-86.893,166.544,45.543,158.307
C09844=1025.999,-116.277,-86.886,166.540,45.545,158.307
C09845=1025.994,-116.527,-86.877,166.538,45.548,158.307
C09846=1025.988,-116.813,-86.867,166.534,45.551,158.307
C09847=1025.981,-117.099,-86.857,166.530,45.555,158.308
C09848=1025.974,-117.384,-86.847,166.527,45.558,158.308
C09849=1025.968,-117.671,-86.837,166.524,45.561,158.308
C09850=1025.962,-117.919,-86.828,166.521,45.563,158.308
C09851=1025.956,-118.170,-86.819,166.518,45.566,158.308
C09852=1025.951,-118.420,-86.811,166.514,45.569,158.308
C09853=1025.945,-118.669,-86.803,166.512,45.571,158.308
C09854=1025.939,-118.919,-86.794,166.509,45.574,158.309
C09855=1025.933,-119.169,-86.786,166.505,45.577,158.309
C09856=1025.928,-119.419,-86.777,166.503,45.580,158.309
C09857=1025.922,-119.669,-86.768,166.499,45.582,158.309
C09858=1025.916,-119.918,-86.760,166.497,45.585,158.309
C09859=1025.911,-120.168,-86.751,166.494,45.588,158.309
C09860=1025.905,-120.418,-86.742,166.490,45.591,158.309
C09861=1025.900,-120.668,-86.734,166.488,45.594,158.310
C09862=1025.894,-120.917,-86.726,166.485,45.596,158.310
C09863=1025.888,-121.167,-86.718,166.482,45.599,158.310
C09864=1025.883,-121.417,-86.709,166.479,45.602,158.310
C09865=1025.877,-121.667,-86.700,166.475,45.605,158.310
C09866=1025.871,-121.917,-86.692,166.473,45.607,158.310
C09867=1025.866,-122.166,-86.684,166.470,45.610,158.311
C09868=1025.860,-122.417,-86.675,166.467,45.612,158.311
C09869=1025.854,-122.666,-86.667,166.464,45.615,158.311
C09870=1025.849,-122.916,-86.659,166.461,45.618,158.311
C09871=1025.844,-123.165,-86.650,166.458,45.621,158.311
C09872=1025.837,-123.416,-86.642,166.455,45.624,158.311
C09873=1025.832,-123.665,-86.633,166.453,45.627,158.311
C09874=1025.826,-123.915,-86.625,166.449,45.629,158.311
C09875=1025.821,-124.165,-86.617,166.446,45.632,158.312
C09876=1025.815,-124.414,-86.609,166.443,45.635,158.312
C09877=1025.809,-124.665,-86.600,166.440,45.638,158.312
C09878=1025.804,-124.915,-86.593,166.438,45.640,158.312
C09879=1025.798,-125.164,-86.584,166.434,45.643,158.312
C09880=1025.793,-125.414,-86.576,166.431,45.646,158.312
C09881=1025.787,-125.663,-86.568,166.429,45.649,158.313
C09882=1025.781,-125.914,-86.559,166.425,45.652,158.313
C09883=1025.775,-126.163,-86.551,166.422,45.654,158.313
C09884=1025.770,-126.413,-86.542,166.419,45.657,158.313
C09885=1025.764,-126.663,-86.535,166.416,45.660,158.313
C09886=1025.759,-126.913,-86.527,166.413,45.663,158.313
C09887=1025.754,-127.162,-86.518,166.410,45.666,158.314
C09888=1025.748,-127.412,-86.510,166.407,45.669,158.314
C09889=1025.742,-127.662,-86.502,166.405,45.672,158.314
C09890=1025.736,-127.911,-86.494,166.401,45.675,158.314
C09891=1025.731,-128.161,-86.486,166.399,45.677,158.314
C09892=1025.727,-128.411,-86.477,166.395,45.679,158.314
C09893=1025.723,-128.660,-86.466,166.392,45.680,158.314
C09894=1025.719,-128.910,-86.457,166.390,45.681,158.314
C09895=1025.716,-129.160,-86.446,166.387,45.682,158.314
C09896=1025.714,-129.409,-86.434,166.385,45.682,158.313
C09897=1025.712,-129.659,-86.423,166.383,45.681,158.313
C09898=1025.710,-129.909,-86.409,166.380,45.680,158.313
C09899=1025.709,-130.159,-86.396,166.378,45.680,158.312
C09900=1025.709,-130.409,-86.382,166.376,45.678,158.312
C09901=1025.709,-130.659,-86.369,166.374,45.675,158.311
C09902=1025.711,-130.908,-86.353,166.372,45.672,158.310
C09903=1025.712,-131.158,-86.338,166.369,45.669,158.310
C09904=1025.714,-131.408,-86.322,166.368,45.666,158.309
C09905=1025.716,-131.658,-86.306,166.367,45.661,158.308
C09906=1025.720,-131.907,-86.288,166.365,45.656,158.307
C09907=1025.723,-132.158,-86.270,166.363,45.651,158.306
C09908=1025.727,-132.407,-86.252,166.362,45.646,158.305
C09909=1025.732,-132.657,-86.234,166.361,45.639,158.304
C09910=1025.429,-132.682,-86.560,166.312,45.907,158.343
C09911=1025.424,-132.433,-86.578,166.314,45.913,158.344
C09912=1025.420,-132.184,-86.597,166.315,45.918,158.346
C09913=1025.417,-131.933,-86.615,166.317,45.924,158.347
C09914=1025.413,-131.683,-86.632,166.319,45.928,158.348
C09915=1025.411,-131.433,-86.649,166.320,45.933,158.348
C09916=1025.409,-131.184,-86.665,166.322,45.937,158.349
C09917=1025.407,-130.934,-86.681,166.324,45.940,158.350
C09918=1025.407,-130.684,-86.696,166.326,45.943,158.351
C09919=1025.406,-130.434,-86.710,166.328,45.945,158.351
C09920=1025.406,-130.184,-86.724,166.330,45.947,158.352
C09921=1025.407,-129.935,-86.737,166.333,45.948,158.352
C09922=1025.409,-129.685,-86.750,166.334,45.949,158.353
C09923=1025.410,-129.435,-86.761,166.336,45.950,158.353
C09924=1025.413,-129.186,-86.773,166.340,45.950,158.354
C09925=1025.416,-128.936,-86.784,166.342,45.949,158.354
C09926=1025.419,-128.686,-86.794,166.345,45.948,158.354
C09927=1025.423,-128.436,-86.804,166.347,45.947,158.354
C09928=1025.428,-128.186,-86.813,166.350,45.944,158.354
C09929=1025.433,-127.937,-86.822,166.353,45.941,158.354
C09930=1025.438,-127.688,-86.829,166.356,45.939,158.354
C09931=1025.444,-127.437,-86.838,166.359,45.936,158.353
C09932=1025.450,-127.188,-86.846,166.363,45.933,158.353
C09933=1025.456,-126.938,-86.854,166.365,45.931,158.353
C09934=1025.461,-126.688,-86.861,166.368,45.928,158.353
C09935=1025.467,-126.439,-86.870,166.372,45.925,158.353
C09936=1025.472,-126.189,-86.878,166.374,45.922,158.353
C09937=1025.478,-125.940,-86.886,166.377,45.919,158.352
C09938=1025.484,-125.689,-86.895,166.381,45.916,158.352
C09939=1025.490,-125.440,-86.903,166.383,45.913,158.352
C09940=1025.495,-125.189,-86.911,166.386,45.910,158.352
C09941=1025.501,-124.940,-86.919,166.390,45.907,158.352
C09942=1025.506,-124.690,-86.927,166.392,45.904,158.352
C09943=1025.512,-124.441,-86.935,166.395,45.901,158.352
C09944=1025.518,-124.190,-86.944,166.399,45.898,158.351
C09945=1025.523,-123.941,-86.952,166.401,45.896,158.351
C09946=1025.528,-123.691,-86.961,166.404,45.893,158.351
C09947=1025.534,-123.442,-86.969,166.406,45.890,158.351
C09948=1025.540,-123.192,-86.977,166.410,45.887,158.351
C09949=1025.545,-122.941,-86.985,166.413,45.884,158.351
C09950=1025.551,-122.691,-86.993,166.416,45.882,158.350
C09951=1025.556,-122.442,-87.002,166.419,45.879,158.350
C09952=1025.562,-122.192,-87.010,166.422,45.876,158.350
C09953=1025.568,-121.942,-87.019,166.425,45.873,158.350
C09954=1025.573,-121.692,-87.027,166.428,45.870,158.350
C09955=1025.579,-121.442,-87.036,166.431,45.867,158.350
C09956=1025.584,-121.193,-87.044,166.434,45.864,158.349
C09957=1025.591,-120.943,-87.052,166.437,45.862,158.350
C09958=1025.596,-120.693,-87.061,166.441,45.859,158.349
C09959=1025.601,-120.443,-87.069,166.443,45.856,158.349
C09960=1025.607,-120.194,-87.078,166.446,45.853,158.349
C09961=1025.613,-119.944,-87.087,166.449,45.850,158.349
C09962=1025.619,-119.694,-87.095,166.452,45.847,158.349
C09963=1025.624,-119.445,-87.104,166.455,45.844,158.349
C09964=1025.629,-119.195,-87.112,166.458,45.842,158.348
C09965=1025.636,-118.945,-87.120,166.461,45.839,158.348
C09966=1025.641,-118.695,-87.129,166.465,45.836,158.348
C09967=1025.646,-118.445,-87.137,166.467,45.834,158.348
C09968=1025.652,-118.195,-87.146,166.470,45.831,158.348
C09969=1025.658,-117.945,-87.154,166.473,45.828,158.348
C09970=1025.664,-117.696,-87.163,166.476,45.825,158.347
C09971=1025.670,-117.410,-87.173,166.479,45.822,158.347
C09972=1025.676,-117.124,-87.183,166.482,45.819,158.347
C09973=1025.683,-116.839,-87.193,166.487,45.815,158.347
C09974=1025.690,-116.553,-87.203,166.490,45.812,158.347
C09975=1025.695,-116.303,-87.211,166.492,45.809,158.347
C09976=1025.701,-116.053,-87.220,166.496,45.806,158.346
C09977=1025.706,-115.803,-87.229,166.499,45.804,158.346
C09978=1025.712,-115.554,-87.237,166.502,45.801,158.346
C09979=1025.719,-115.304,-87.246,166.505,45.798,158.346
C09980=1025.724,-115.054,-87.255,166.508,45.795,158.346
C09981=1025.729,-114.805,-87.263,166.510,45.792,158.346
C09982=1025.735,-114.554,-87.272,166.514,45.789,158.346
C09983=1025.741,-114.305,-87.281,166.516,45.787,158.346
C09984=1025.746,-114.055,-87.290,166.520,45.784,158.345
C09985=1025.752,-113.805,-87.298,166.523,45.781,158.345
C09986=1025.757,-113.556,-87.308,166.525,45.779,158.345
C09987=1025.763,-113.305,-87.317,166.529,45.776,158.345
C09988=1025.768,-113.056,-87.325,166.532,45.773,158.345
C09989=1025.775,-112.806,-87.334,166.535,45.771,158.345
C09990=1025.781,-112.557,-87.342,166.538,45.768,158.345
C09991=1025.786,-112.306,-87.351,166.540,45.765,158.344
C09992=1025.792,-112.057,-87.361,166.544,45.763,158.344
C09993=1025.797,-111.807,-87.369,166.547,45.760,158.344
C09994=1025.803,-111.558,-87.379,166.550,45.757,158.344
C09995=1025.809,-111.308,-87.387,166.553,45.754,158.344
C09996=1025.815,-111.057,-87.396,166.555,45.751,158.344
//INST
///DATE 2021/06/17 10:58
///ATTR SC,RW,RJ
////FRAME ROBOT
///GROUP1 RB1
NOP
MOVL C00000 V=800.0 PL=0
MOVL C00001 V=800.0 PL=0
MOVL C00002 V=800.0 PL=0
MOVL C00003 V=800.0 PL=0
MOVL C00004 V=800.0 PL=0
MOVL C00005 V=800.0 PL=0
MOVL C00006 V=800.0 PL=0
MOVL C00007 V=800.0 PL=0
MOVL C00008 V=800.0 PL=0
MOVL C00009 V=800.0 PL=0
MOVL C00010 V=800.0 PL=0
MOVL C00011 V=800.0 PL=0
MOVL C00012 V=800.0 PL=0
MOVL C00013 V=800.0 PL=0
MOVL C00014 V=800.0 PL=0
MOVL C00015 V=800.0 PL=0
MOVL C00016 V=800.0 PL=0
MOVL C00017 V=800.0 PL=0
MOVL C00018 V=800.0 PL=0
MOVL C00019 V=800.0 PL=0
MOVL C00020 V=800.0 PL=0
MOVL C00021 V=800.0 PL=0
MOVL C00022 V=800.0 PL=0
MOVL C00023 V=800.0 PL=0
MOVL C00024 V=800.0 PL=0
MOVL C00025 V=800.0 PL=0
MOVL C00026 V=800.0 PL=0
MOVL C00027 V=800.0 PL=0
MOVL C00028 V=800.0 PL=0
MOVL C00029 V=800.0 PL=0
MOVL C00030 V=800.0 PL=0
MOVL C00031 V=800.0 PL=0
MOVL C00032 V=800.0 PL=0
MOVL C00033 V=800.0 PL=0
MOVL C00034 V=800.0 PL=0
MOVL C00035 V=800.0 PL=0
MOVL C00036 V=800.0 PL=0
MOVL C00037 V=800.0 PL=0
MOVL C00038 V=800.0 PL=0
MOVL C00039 V=800.0 PL=0
MOVL C00040 V=800.0 PL=0
MOVL C00041 V=800.0 PL=0
MOVL C00042 V=800.0 PL=0
MOVL C00043 V=800.0 PL=0
MOVL C00044 V=800.0 PL=0
MOVL C00045 V=800.0 PL=0
MOVL C00046 V=800.0 PL=0
MOVL C00047 V=800.0 PL=0
MOVL C00048 V=800.0 PL=0
MOVL C00049 V=800.0 PL=0
MOVL C00050 V=800.0 PL=0
MOVL C00051 V=800.0 PL=0
MOVL C00052 V=800.0 PL=0
MOVL C00053 V=800.0 PL=0
MOVL C00054 V=800.0 PL=0
MOVL C00055 V=800.0 PL=0
MOVL C00056 V=800.0 PL=0
MOVL C00057 V=800.0 PL=0
MOVL C00058 V=800.0 PL=0
MOVL C00059 V=800.0 PL=0
MOVL C00060 V=800.0 PL=0
MOVL C00061 V=800.0 PL=0
MOVL C00062 V=800.0 PL=0
MOVL C00063 V=800.0 PL=0
MOVL C00064 V=800.0 PL=0
MOVL C00065 V=800.0 PL=0
MOVL C00066 V=800.0 PL=0
MOVL C00067 V=800.0 PL=0
MOVL C00068 V=800.0 PL=0
MOVL C00069 V=800.0 PL=0
MOVL C00070 V=800.0 PL=0
MOVL C00071 V=800.0 PL=0
MOVL C00072 V=800.0 PL=0
MOVL C00073 V=800.0 PL=0
MOVL C00074 V=800.0 PL=0
MOVL C00075 V=800.0 PL=0
MOVL C00076 V=800.0 PL=0
MOVL C00077 V=800.0 PL=0
MOVL C00078 V=800.0 PL=0
MOVL C00079 V=800.0 PL=0
MOVL C00080 V=800.0 PL=0
MOVL C00081 V=800.0 PL=0
MOVL C00082 V=800.0 PL=0
MOVL C00083 V=800.0 PL=0
MOVL C00084 V=800.0 PL=0
MOVL C00085 V=800.0 PL=0
MOVL C00086 V=800.0 PL=0
MOVL C00087 V=800.0 PL=0
MOVL C00088 V=800.0 PL=0
MOVL C00089 V=800.0 PL=0
MOVL C00090 V=800.0 PL=0
MOVL C00091 V=800.0 PL=0
MOVL C00092 V=800.0 PL=0
MOVL C00093 V=800.0 PL=0
MOVL C00094 V=800.0 PL=0
MOVL C00095 V=800.0 PL=0
MOVL C00096 V=800.0 PL=0
MOVL C00097 V=800.0 PL=0
MOVL C00098 V=800.0 PL=0
MOVL C00099 V=800.0 PL=0
MOVL C00100 V=800.0 PL=0
MOVL C00101 V=800.0 PL=0
MOVL C00102 V=800.0 PL=0
MOVL C00103 V=800.0 PL=0
MOVL C00104 V=800.0 PL=0
MOVL C00105 V=800.0 PL=0
MOVL C00106 V=800.0 PL=0
MOVL C00107 V=800.0 PL=0
MOVL C00108 V=800.0 PL=0
MOVL C00109 V=800.0 PL=0
MOVL C00110 V=800.0 PL=0
MOVL C00111 V=800.0 PL=0
MOVL C00112 V=800.0 PL=0
MOVL C00113 V=800.0 PL=0
MOVL C00114 V=800.0 PL=0
MOVL C00115 V=800.0 PL=0
MOVL C00116 V=800.0 PL=0
MOVL C00117 V=800.0 PL=0
MOVL C00118 V=800.0 PL=0
MOVL C00119 V=800.0 PL=0
MOVL C00120 V=800.0 PL=0
MOVL C00121 V=800.0 PL=0
MOVL C00122 V=800.0 PL=0
MOVL C00123 V=800.0 PL=0
MOVL C00124 V=800.0 PL=0
MOVL C00125 V=800.0 PL=0
MOVL C00126 V=800.0 PL=0
MOVL C00127 V=800.0 PL=0
MOVL C00128 V=800.0 PL=0
MOVL C00129 V=800.0 PL=0
MOVL C00130 V=800.0 PL=0
MOVL C00131 V=800.0 PL=0
MOVL C00132 V=800.0 PL=0
MOVL C00133 V=800.0 PL=0
MOVL C00134 V=800.0 PL=0
MOVL C00135 V=800.0 PL=0
MOVL C00136 V=800.0 PL=0
MOVL C00137 V=800.0 PL=0
MOVL C00138 V=800.0 PL=0
MOVL C00139 V=800.0 PL=0
MOVL C00140 V=800.0 PL=0
MOVL C00141 V=800.0 PL=0
MOVL C00142 V=800.0 PL=0
MOVL C00143 V=800.0 PL=0
MOVL C00144 V=800.0 PL=0
MOVL C00145 V=800.0 PL=0
MOVL C00146 V=800.0 PL=0
MOVL C00147 V=800.0 PL=0
MOVL C00148 V=800.0 PL=0
MOVL C00149 V=800.0 PL=0
MOVL C00150 V=800.0 PL=0
MOVL C00151 V=800.0 PL=0
MOVL C00152 V=800.0 PL=0
MOVL C00153 V=800.0 PL=0
MOVL C00154 V=800.0 PL=0
MOVL C00155 V=800.0 PL=0
MOVL C00156 V=800.0 PL=0
MOVL C00157 V=800.0 PL=0
MOVL C00158 V=800.0 PL=0
MOVL C00159 V=800.0 PL=0
MOVL C00160 V=800.0 PL=0
MOVL C00161 V=800.0 PL=0
MOVL C00162 V=800.0 PL=0
MOVL C00163 V=800.0 PL=0
MOVL C00164 V=800.0 PL=0
MOVL C00165 V=800.0 PL=0
MOVL C00166 V=800.0 PL=0
MOVL C00167 V=800.0 PL=0
MOVL C00168 V=800.0 PL=0
MOVL C00169 V=800.0 PL=0
MOVL C00170 V=800.0 PL=0
MOVL C00171 V=800.0 PL=0
MOVL C00172 V=800.0 PL=0
MOVL C00173 V=800.0 PL=0
MOVL C00174 V=800.0 PL=0
MOVL C00175 V=800.0 PL=0
MOVL C00176 V=800.0 PL=0
MOVL C00177 V=800.0 PL=0
MOVL C00178 V=800.0 PL=0
MOVL C00179 V=800.0 PL=0
MOVL C00180 V=800.0 PL=0
MOVL C00181 V=800.0 PL=0
MOVL C00182 V=800.0 PL=0
MOVL C00183 V=800.0 PL=0
MOVL C00184 V=800.0 PL=0
MOVL C00185 V=800.0 PL=0
MOVL C00186 V=800.0 PL=0
MOVL C00187 V=800.0 PL=0
MOVL C00188 V=800.0 PL=0
MOVL C00189 V=800.0 PL=0
MOVL C00190 V=800.0 PL=0
MOVL C00191 V=800.0 PL=0
MOVL C00192 V=800.0 PL=0
MOVL C00193 V=800.0 PL=0
MOVL C00194 V=800.0 PL=0
MOVL C00195 V=800.0 PL=0
MOVL C00196 V=800.0 PL=0
MOVL C00197 V=800.0 PL=0
MOVL C00198 V=800.0 PL=0
MOVL C00199 V=800.0 PL=0
MOVL C00200 V=800.0 PL=0
MOVL C00201 V=800.0 PL=0
MOVL C00202 V=800.0 PL=0
MOVL C00203 V=800.0 PL=0
MOVL C00204 V=800.0 PL=0
MOVL C00205 V=800.0 PL=0
MOVL C00206 V=800.0 PL=0
MOVL C00207 V=800.0 PL=0
MOVL C00208 V=800.0 PL=0
MOVL C00209 V=800.0 PL=0
MOVL C00210 V=800.0 PL=0
MOVL C00211 V=800.0 PL=0
MOVL C00212 V=800.0 PL=0
MOVL C00213 V=800.0 PL=0
MOVL C00214 V=800.0 PL=0
MOVL C00215 V=800.0 PL=0
MOVL C00216 V=800.0 PL=0
MOVL C00217 V=800.0 PL=0
MOVL C00218 V=800.0 PL=0
MOVL C00219 V=800.0 PL=0
MOVL C00220 V=800.0 PL=0
MOVL C00221 V=800.0 PL=0
MOVL C00222 V=800.0 PL=0
MOVL C00223 V=800.0 PL=0
MOVL C00224 V=800.0 PL=0
MOVL C00225 V=800.0 PL=0
MOVL C00226 V=800.0 PL=0
MOVL C00227 V=800.0 PL=0
MOVL C00228 V=800.0 PL=0
MOVL C00229 V=800.0 PL=0
MOVL C00230 V=800.0 PL=0
MOVL C00231 V=800.0 PL=0
MOVL C00232 V=800.0 PL=0
MOVL C00233 V=800.0 PL=0
MOVL C00234 V=800.0 PL=0
MOVL C00235 V=800.0 PL=0
MOVL C00236 V=800.0 PL=0
MOVL C00237 V=800.0 PL=0
MOVL C00238 V=800.0 PL=0
MOVL C00239 V=800.0 PL=0
MOVL C00240 V=800.0 PL=0
MOVL C00241 V=800.0 PL=0
MOVL C00242 V=800.0 PL=0
MOVL C00243 V=800.0 PL=0
MOVL C00244 V=800.0 PL=0
MOVL C00245 V=800.0 PL=0
MOVL C00246 V=800.0 PL=0
MOVL C00247 V=800.0 PL=0
MOVL C00248 V=800.0 PL=0
MOVL C00249 V=800.0 PL=0
MOVL C00250 V=800.0 PL=0
MOVL C00251 V=800.0 PL=0
MOVL C00252 V=800.0 PL=0
MOVL C00253 V=800.0 PL=0
MOVL C00254 V=800.0 PL=0
MOVL C00255 V=800.0 PL=0
MOVL C00256 V=800.0 PL=0
MOVL C00257 V=800.0 PL=0
MOVL C00258 V=800.0 PL=0
MOVL C00259 V=800.0 PL=0
MOVL C00260 V=800.0 PL=0
MOVL C00261 V=800.0 PL=0
MOVL C00262 V=800.0 PL=0
MOVL C00263 V=800.0 PL=0
MOVL C00264 V=800.0 PL=0
MOVL C00265 V=800.0 PL=0
MOVL C00266 V=800.0 PL=0
MOVL C00267 V=800.0 PL=0
MOVL C00268 V=800.0 PL=0
MOVL C00269 V=800.0 PL=0
MOVL C00270 V=800.0 PL=0
MOVL C00271 V=800.0 PL=0
MOVL C00272 V=800.0 PL=0
MOVL C00273 V=800.0 PL=0
MOVL C00274 V=800.0 PL=0
MOVL C00275 V=800.0 PL=0
MOVL C00276 V=800.0 PL=0
MOVL C00277 V=800.0 PL=0
MOVL C00278 V=800.0 PL=0
MOVL C00279 V=800.0 PL=0
MOVL C00280 V=800.0 PL=0
MOVL C00281 V=800.0 PL=0
MOVL C00282 V=800.0 PL=0
MOVL C00283 V=800.0 PL=0
MOVL C00284 V=800.0 PL=0
MOVL C00285 V=800.0 PL=0
MOVL C00286 V=800.0 PL=0
MOVL C00287 V=800.0 PL=0
MOVL C00288 V=800.0 PL=0
MOVL C00289 V=800.0 PL=0
MOVL C00290 V=800.0 PL=0
MOVL C00291 V=800.0 PL=0
MOVL C00292 V=800.0 PL=0
MOVL C00293 V=800.0 PL=0
MOVL C00294 V=800.0 PL=0
MOVL C00295 V=800.0 PL=0
MOVL C00296 V=800.0 PL=0
MOVL C00297 V=800.0 PL=0
MOVL C00298 V=800.0 PL=0
MOVL C00299 V=800.0 PL=0
MOVL C00300 V=800.0 PL=0
MOVL C00301 V=800.0 PL=0
MOVL C00302 V=800.0 PL=0
MOVL C00303 V=800.0 PL=0
MOVL C00304 V=800.0 PL=0
MOVL C00305 V=800.0 PL=0
MOVL C00306 V=800.0 PL=0
MOVL C00307 V=800.0 PL=0
MOVL C00308 V=800.0 PL=0
MOVL C00309 V=800.0 PL=0
MOVL C00310 V=800.0 PL=0
MOVL C00311 V=800.0 PL=0
MOVL C00312 V=800.0 PL=0
MOVL C00313 V=800.0 PL=0
MOVL C00314 V=800.0 PL=0
MOVL C00315 V=800.0 PL=0
MOVL C00316 V=800.0 PL=0
MOVL C00317 V=800.0 PL=0
MOVL C00318 V=800.0 PL=0
MOVL C00319 V=800.0 PL=0
MOVL C00320 V=800.0 PL=0
MOVL C00321 V=800.0 PL=0
MOVL C00322 V=800.0 PL=0
MOVL C00323 V=800.0 PL=0
MOVL C00324 V=800.0 PL=0
MOVL C00325 V=800.0 PL=0
MOVL C00326 V=800.0 PL=0
MOVL C00327 V=800.0 PL=0
MOVL C00328 V=800.0 PL=0
MOVL C00329 V=800.0 PL=0
MOVL C00330 V=800.0 PL=0
MOVL C00331 V=800.0 PL=0
MOVL C00332 V=800.0 PL=0
MOVL C00333 V=800.0 PL=0
MOVL C00334 V=800.0 PL=0
MOVL C00335 V=800.0 PL=0
MOVL C00336 V=800.0 PL=0
MOVL C00337 V=800.0 PL=0
MOVL C00338 V=800.0 PL=0
MOVL C00339 V=800.0 PL=0
MOVL C00340 V=800.0 PL=0
MOVL C00341 V=800.0 PL=0
MOVL C00342 V=800.0 PL=0
MOVL C00343 V=800.0 PL=0
MOVL C00344 V=800.0 PL=0
MOVL C00345 V=800.0 PL=0
MOVL C00346 V=800.0 PL=0
MOVL C00347 V=800.0 PL=0
MOVL C00348 V=800.0 PL=0
MOVL C00349 V=800.0 PL=0
MOVL C00350 V=800.0 PL=0
MOVL C00351 V=800.0 PL=0
MOVL C00352 V=800.0 PL=0
MOVL C00353 V=800.0 PL=0
MOVL C00354 V=800.0 PL=0
MOVL C00355 V=800.0 PL=0
MOVL C00356 V=800.0 PL=0
MOVL C00357 V=800.0 PL=0
MOVL C00358 V=800.0 PL=0
MOVL C00359 V=800.0 PL=0
MOVL C00360 V=800.0 PL=0
MOVL C00361 V=800.0 PL=0
MOVL C00362 V=800.0 PL=0
MOVL C00363 V=800.0 PL=0
MOVL C00364 V=800.0 PL=0
MOVL C00365 V=800.0 PL=0
MOVL C00366 V=800.0 PL=0
MOVL C00367 V=800.0 PL=0
MOVL C00368 V=800.0 PL=0
MOVL C00369 V=800.0 PL=0
MOVL C00370 V=800.0 PL=0
MOVL C00371 V=800.0 PL=0
MOVL C00372 V=800.0 PL=0
MOVL C00373 V=800.0 PL=0
MOVL C00374 V=800.0 PL=0
MOVL C00375 V=800.0 PL=0
MOVL C00376 V=800.0 PL=0
MOVL C00377 V=800.0 PL=0
MOVL C00378 V=800.0 PL=0
MOVL C00379 V=800.0 PL=0
MOVL C00380 V=800.0 PL=0
MOVL C00381 V=800.0 PL=0
MOVL C00382 V=800.0 PL=0
MOVL C00383 V=800.0 PL=0
MOVL C00384 V=800.0 PL=0
MOVL C00385 V=800.0 PL=0
MOVL C00386 V=800.0 PL=0
MOVL C00387 V=800.0 PL=0
MOVL C00388 V=800.0 PL=0
MOVL C00389 V=800.0 PL=0
MOVL C00390 V=800.0 PL=0
MOVL C00391 V=800.0 PL=0
MOVL C00392 V=800.0 PL=0
MOVL C00393 V=800.0 PL=0
MOVL C00394 V=800.0 PL=0
MOVL C00395 V=800.0 PL=0
MOVL C00396 V=800.0 PL=0
MOVL C00397 V=800.0 PL=0
MOVL C00398 V=800.0 PL=0
MOVL C00399 V=800.0 PL=0
MOVL C00400 V=800.0 PL=0
MOVL C00401 V=800.0 PL=0
MOVL C00402 V=800.0 PL=0
MOVL C00403 V=800.0 PL=0
MOVL C00404 V=800.0 PL=0
MOVL C00405 V=800.0 PL=0
MOVL C00406 V=800.0 PL=0
MOVL C00407 V=800.0 PL=0
MOVL C00408 V=800.0 PL=0
MOVL C00409 V=800.0 PL=0
MOVL C00410 V=800.0 PL=0
MOVL C00411 V=800.0 PL=0
MOVL C00412 V=800.0 PL=0
MOVL C00413 V=800.0 PL=0
MOVL C00414 V=800.0 PL=0
MOVL C00415 V=800.0 PL=0
MOVL C00416 V=800.0 PL=0
MOVL C00417 V=800.0 PL=0
MOVL C00418 V=800.0 PL=0
MOVL C00419 V=800.0 PL=0
MOVL C00420 V=800.0 PL=0
MOVL C00421 V=800.0 PL=0
MOVL C00422 V=800.0 PL=0
MOVL C00423 V=800.0 PL=0
MOVL C00424 V=800.0 PL=0
MOVL C00425 V=800.0 PL=0
MOVL C00426 V=800.0 PL=0
MOVL C00427 V=800.0 PL=0
MOVL C00428 V=800.0 PL=0
MOVL C00429 V=800.0 PL=0
MOVL C00430 V=800.0 PL=0
MOVL C00431 V=800.0 PL=0
MOVL C00432 V=800.0 PL=0
MOVL C00433 V=800.0 PL=0
MOVL C00434 V=800.0 PL=0
MOVL C00435 V=800.0 PL=0
MOVL C00436 V=800.0 PL=0
MOVL C00437 V=800.0 PL=0
MOVL C00438 V=800.0 PL=0
MOVL C00439 V=800.0 PL=0
MOVL C00440 V=800.0 PL=0
MOVL C00441 V=800.0 PL=0
MOVL C00442 V=800.0 PL=0
MOVL C00443 V=800.0 PL=0
MOVL C00444 V=800.0 PL=0
MOVL C00445 V=800.0 PL=0
MOVL C00446 V=800.0 PL=0
MOVL C00447 V=800.0 PL=0
MOVL C00448 V=800.0 PL=0
MOVL C00449 V=800.0 PL=0
MOVL C00450 V=800.0 PL=0
MOVL C00451 V=800.0 PL=0
MOVL C00452 V=800.0 PL=0
MOVL C00453 V=800.0 PL=0
MOVL C00454 V=800.0 PL=0
MOVL C00455 V=800.0 PL=0
MOVL C00456 V=800.0 PL=0
MOVL C00457 V=800.0 PL=0
MOVL C00458 V=800.0 PL=0
MOVL C00459 V=800.0 PL=0
MOVL C00460 V=800.0 PL=0
MOVL C00461 V=800.0 PL=0
MOVL C00462 V=800.0 PL=0
MOVL C00463 V=800.0 PL=0
MOVL C00464 V=800.0 PL=0
MOVL C00465 V=800.0 PL=0
MOVL C00466 V=800.0 PL=0
MOVL C00467 V=800.0 PL=0
MOVL C00468 V=800.0 PL=0
MOVL C00469 V=800.0 PL=0
MOVL C00470 V=800.0 PL=0
MOVL C00471 V=800.0 PL=0
MOVL C00472 V=800.0 PL=0
MOVL C00473 V=800.0 PL=0
MOVL C00474 V=800.0 PL=0
MOVL C00475 V=800.0 PL=0
MOVL C00476 V=800.0 PL=0
MOVL C00477 V=800.0 PL=0
MOVL C00478 V=800.0 PL=0
MOVL C00479 V=800.0 PL=0
MOVL C00480 V=800.0 PL=0
MOVL C00481 V=800.0 PL=0
MOVL C00482 V=800.0 PL=0
MOVL C00483 V=800.0 PL=0
MOVL C00484 V=800.0 PL=0
MOVL C00485 V=800.0 PL=0
MOVL C00486 V=800.0 PL=0
MOVL C00487 V=800.0 PL=0
MOVL C00488 V=800.0 PL=0
MOVL C00489 V=800.0 PL=0
MOVL C00490 V=800.0 PL=0
MOVL C00491 V=800.0 PL=0
MOVL C00492 V=800.0 PL=0
MOVL C00493 V=800.0 PL=0
MOVL C00494 V=800.0 PL=0
MOVL C00495 V=800.0 PL=0
MOVL C00496 V=800.0 PL=0
MOVL C00497 V=800.0 PL=0
MOVL C00498 V=800.0 PL=0
MOVL C00499 V=800.0 PL=0
MOVL C00500 V=800.0 PL=0
MOVL C00501 V=800.0 PL=0
MOVL C00502 V=800.0 PL=0
MOVL C00503 V=800.0 PL=0
MOVL C00504 V=800.0 PL=0
MOVL C00505 V=800.0 PL=0
MOVL C00506 V=800.0 PL=0
MOVL C00507 V=800.0 PL=0
MOVL C00508 V=800.0 PL=0
MOVL C00509 V=800.0 PL=0
MOVL C00510 V=800.0 PL=0
MOVL C00511 V=800.0 PL=0
MOVL C00512 V=800.0 PL=0
MOVL C00513 V=800.0 PL=0
MOVL C00514 V=800.0 PL=0
MOVL C00515 V=800.0 PL=0
MOVL C00516 V=800.0 PL=0
MOVL C00517 V=800.0 PL=0
MOVL C00518 V=800.0 PL=0
MOVL C00519 V=800.0 PL=0
MOVL C00520 V=800.0 PL=0
MOVL C00521 V=800.0 PL=0
MOVL C00522 V=800.0 PL=0
MOVL C00523 V=800.0 PL=0
MOVL C00524 V=800.0 PL=0
MOVL C00525 V=800.0 PL=0
MOVL C00526 V=800.0 PL=0
MOVL C00527 V=800.0 PL=0
MOVL C00528 V=800.0 PL=0
MOVL C00529 V=800.0 PL=0
MOVL C00530 V=800.0 PL=0
MOVL C00531 V=800.0 PL=0
MOVL C00532 V=800.0 PL=0
MOVL C00533 V=800.0 PL=0
MOVL C00534 V=800.0 PL=0
MOVL C00535 V=800.0 PL=0
MOVL C00536 V=800.0 PL=0
MOVL C00537 V=800.0 PL=0
MOVL C00538 V=800.0 PL=0
MOVL C00539 V=800.0 PL=0
MOVL C00540 V=800.0 PL=0
MOVL C00541 V=800.0 PL=0
MOVL C00542 V=800.0 PL=0
MOVL C00543 V=800.0 PL=0
MOVL C00544 V=800.0 PL=0
MOVL C00545 V=800.0 PL=0
MOVL C00546 V=800.0 PL=0
MOVL C00547 V=800.0 PL=0
MOVL C00548 V=800.0 PL=0
MOVL C00549 V=800.0 PL=0
MOVL C00550 V=800.0 PL=0
MOVL C00551 V=800.0 PL=0
MOVL C00552 V=800.0 PL=0
MOVL C00553 V=800.0 PL=0
MOVL C00554 V=800.0 PL=0
MOVL C00555 V=800.0 PL=0
MOVL C00556 V=800.0 PL=0
MOVL C00557 V=800.0 PL=0
MOVL C00558 V=800.0 PL=0
MOVL C00559 V=800.0 PL=0
MOVL C00560 V=800.0 PL=0
MOVL C00561 V=800.0 PL=0
MOVL C00562 V=800.0 PL=0
MOVL C00563 V=800.0 PL=0
MOVL C00564 V=800.0 PL=0
MOVL C00565 V=800.0 PL=0
MOVL C00566 V=800.0 PL=0
MOVL C00567 V=800.0 PL=0
MOVL C00568 V=800.0 PL=0
MOVL C00569 V=800.0 PL=0
MOVL C00570 V=800.0 PL=0
MOVL C00571 V=800.0 PL=0
MOVL C00572 V=800.0 PL=0
MOVL C00573 V=800.0 PL=0
MOVL C00574 V=800.0 PL=0
MOVL C00575 V=800.0 PL=0
MOVL C00576 V=800.0 PL=0
MOVL C00577 V=800.0 PL=0
MOVL C00578 V=800.0 PL=0
MOVL C00579 V=800.0 PL=0
MOVL C00580 V=800.0 PL=0
MOVL C00581 V=800.0 PL=0
MOVL C00582 V=800.0 PL=0
MOVL C00583 V=800.0 PL=0
MOVL C00584 V=800.0 PL=0
MOVL C00585 V=800.0 PL=0
MOVL C00586 V=800.0 PL=0
MOVL C00587 V=800.0 PL=0
MOVL C00588 V=800.0 PL=0
MOVL C00589 V=800.0 PL=0
MOVL C00590 V=800.0 PL=0
MOVL C00591 V=800.0 PL=0
MOVL C00592 V=800.0 PL=0
MOVL C00593 V=800.0 PL=0
MOVL C00594 V=800.0 PL=0
MOVL C00595 V=800.0 PL=0
MOVL C00596 V=800.0 PL=0
MOVL C00597 V=800.0 PL=0
MOVL C00598 V=800.0 PL=0
MOVL C00599 V=800.0 PL=0
MOVL C00600 V=800.0 PL=0
MOVL C00601 V=800.0 PL=0
MOVL C00602 V=800.0 PL=0
MOVL C00603 V=800.0 PL=0
MOVL C00604 V=800.0 PL=0
MOVL C00605 V=800.0 PL=0
MOVL C00606 V=800.0 PL=0
MOVL C00607 V=800.0 PL=0
MOVL C00608 V=800.0 PL=0
MOVL C00609 V=800.0 PL=0
MOVL C00610 V=800.0 PL=0
MOVL C00611 V=800.0 PL=0
MOVL C00612 V=800.0 PL=0
MOVL C00613 V=800.0 PL=0
MOVL C00614 V=800.0 PL=0
MOVL C00615 V=800.0 PL=0
MOVL C00616 V=800.0 PL=0
MOVL C00617 V=800.0 PL=0
MOVL C00618 V=800.0 PL=0
MOVL C00619 V=800.0 PL=0
MOVL C00620 V=800.0 PL=0
MOVL C00621 V=800.0 PL=0
MOVL C00622 V=800.0 PL=0
MOVL C00623 V=800.0 PL=0
MOVL C00624 V=800.0 PL=0
MOVL C00625 V=800.0 PL=0
MOVL C00626 V=800.0 PL=0
MOVL C00627 V=800.0 PL=0
MOVL C00628 V=800.0 PL=0
MOVL C00629 V=800.0 PL=0
MOVL C00630 V=800.0 PL=0
MOVL C00631 V=800.0 PL=0
MOVL C00632 V=800.0 PL=0
MOVL C00633 V=800.0 PL=0
MOVL C00634 V=800.0 PL=0
MOVL C00635 V=800.0 PL=0
MOVL C00636 V=800.0 PL=0
MOVL C00637 V=800.0 PL=0
MOVL C00638 V=800.0 PL=0
MOVL C00639 V=800.0 PL=0
MOVL C00640 V=800.0 PL=0
MOVL C00641 V=800.0 PL=0
MOVL C00642 V=800.0 PL=0
MOVL C00643 V=800.0 PL=0
MOVL C00644 V=800.0 PL=0
MOVL C00645 V=800.0 PL=0
MOVL C00646 V=800.0 PL=0
MOVL C00647 V=800.0 PL=0
MOVL C00648 V=800.0 PL=0
MOVL C00649 V=800.0 PL=0
MOVL C00650 V=800.0 PL=0
MOVL C00651 V=800.0 PL=0
MOVL C00652 V=800.0 PL=0
MOVL C00653 V=800.0 PL=0
MOVL C00654 V=800.0 PL=0
MOVL C00655 V=800.0 PL=0
MOVL C00656 V=800.0 PL=0
MOVL C00657 V=800.0 PL=0
MOVL C00658 V=800.0 PL=0
MOVL C00659 V=800.0 PL=0
MOVL C00660 V=800.0 PL=0
MOVL C00661 V=800.0 PL=0
MOVL C00662 V=800.0 PL=0
MOVL C00663 V=800.0 PL=0
MOVL C00664 V=800.0 PL=0
MOVL C00665 V=800.0 PL=0
MOVL C00666 V=800.0 PL=0
MOVL C00667 V=800.0 PL=0
MOVL C00668 V=800.0 PL=0
MOVL C00669 V=800.0 PL=0
MOVL C00670 V=800.0 PL=0
MOVL C00671 V=800.0 PL=0
MOVL C00672 V=800.0 PL=0
MOVL C00673 V=800.0 PL=0
MOVL C00674 V=800.0 PL=0
MOVL C00675 V=800.0 PL=0
MOVL C00676 V=800.0 PL=0
MOVL C00677 V=800.0 PL=0
MOVL C00678 V=800.0 PL=0
MOVL C00679 V=800.0 PL=0
MOVL C00680 V=800.0 PL=0
MOVL C00681 V=800.0 PL=0
MOVL C00682 V=800.0 PL=0
MOVL C00683 V=800.0 PL=0
MOVL C00684 V=800.0 PL=0
MOVL C00685 V=800.0 PL=0
MOVL C00686 V=800.0 PL=0
MOVL C00687 V=800.0 PL=0
MOVL C00688 V=800.0 PL=0
MOVL C00689 V=800.0 PL=0
MOVL C00690 V=800.0 PL=0
MOVL C00691 V=800.0 PL=0
MOVL C00692 V=800.0 PL=0
MOVL C00693 V=800.0 PL=0
MOVL C00694 V=800.0 PL=0
MOVL C00695 V=800.0 PL=0
MOVL C00696 V=800.0 PL=0
MOVL C00697 V=800.0 PL=0
MOVL C00698 V=800.0 PL=0
MOVL C00699 V=800.0 PL=0
MOVL C00700 V=800.0 PL=0
MOVL C00701 V=800.0 PL=0
MOVL C00702 V=800.0 PL=0
MOVL C00703 V=800.0 PL=0
MOVL C00704 V=800.0 PL=0
MOVL C00705 V=800.0 PL=0
MOVL C00706 V=800.0 PL=0
MOVL C00707 V=800.0 PL=0
MOVL C00708 V=800.0 PL=0
MOVL C00709 V=800.0 PL=0
MOVL C00710 V=800.0 PL=0
MOVL C00711 V=800.0 PL=0
MOVL C00712 V=800.0 PL=0
MOVL C00713 V=800.0 PL=0
MOVL C00714 V=800.0 PL=0
MOVL C00715 V=800.0 PL=0
MOVL C00716 V=800.0 PL=0
MOVL C00717 V=800.0 PL=0
MOVL C00718 V=800.0 PL=0
MOVL C00719 V=800.0 PL=0
MOVL C00720 V=800.0 PL=0
MOVL C00721 V=800.0 PL=0
MOVL C00722 V=800.0 PL=0
MOVL C00723 V=800.0 PL=0
MOVL C00724 V=800.0 PL=0
MOVL C00725 V=800.0 PL=0
MOVL C00726 V=800.0 PL=0
MOVL C00727 V=800.0 PL=0
MOVL C00728 V=800.0 PL=0
MOVL C00729 V=800.0 PL=0
MOVL C00730 V=800.0 PL=0
MOVL C00731 V=800.0 PL=0
MOVL C00732 V=800.0 PL=0
MOVL C00733 V=800.0 PL=0
MOVL C00734 V=800.0 PL=0
MOVL C00735 V=800.0 PL=0
MOVL C00736 V=800.0 PL=0
MOVL C00737 V=800.0 PL=0
MOVL C00738 V=800.0 PL=0
MOVL C00739 V=800.0 PL=0
MOVL C00740 V=800.0 PL=0
MOVL C00741 V=800.0 PL=0
MOVL C00742 V=800.0 PL=0
MOVL C00743 V=800.0 PL=0
MOVL C00744 V=800.0 PL=0
MOVL C00745 V=800.0 PL=0
MOVL C00746 V=800.0 PL=0
MOVL C00747 V=800.0 PL=0
MOVL C00748 V=800.0 PL=0
MOVL C00749 V=800.0 PL=0
MOVL C00750 V=800.0 PL=0
MOVL C00751 V=800.0 PL=0
MOVL C00752 V=800.0 PL=0
MOVL C00753 V=800.0 PL=0
MOVL C00754 V=800.0 PL=0
MOVL C00755 V=800.0 PL=0
MOVL C00756 V=800.0 PL=0
MOVL C00757 V=800.0 PL=0
MOVL C00758 V=800.0 PL=0
MOVL C00759 V=800.0 PL=0
MOVL C00760 V=800.0 PL=0
MOVL C00761 V=800.0 PL=0
MOVL C00762 V=800.0 PL=0
MOVL C00763 V=800.0 PL=0
MOVL C00764 V=800.0 PL=0
MOVL C00765 V=800.0 PL=0
MOVL C00766 V=800.0 PL=0
MOVL C00767 V=800.0 PL=0
MOVL C00768 V=800.0 PL=0
MOVL C00769 V=800.0 PL=0
MOVL C00770 V=800.0 PL=0
MOVL C00771 V=800.0 PL=0
MOVL C00772 V=800.0 PL=0
MOVL C00773 V=800.0 PL=0
MOVL C00774 V=800.0 PL=0
MOVL C00775 V=800.0 PL=0
MOVL C00776 V=800.0 PL=0
MOVL C00777 V=800.0 PL=0
MOVL C00778 V=800.0 PL=0
MOVL C00779 V=800.0 PL=0
MOVL C00780 V=800.0 PL=0
MOVL C00781 V=800.0 PL=0
MOVL C00782 V=800.0 PL=0
MOVL C00783 V=800.0 PL=0
MOVL C00784 V=800.0 PL=0
MOVL C00785 V=800.0 PL=0
MOVL C00786 V=800.0 PL=0
MOVL C00787 V=800.0 PL=0
MOVL C00788 V=800.0 PL=0
MOVL C00789 V=800.0 PL=0
MOVL C00790 V=800.0 PL=0
MOVL C00791 V=800.0 PL=0
MOVL C00792 V=800.0 PL=0
MOVL C00793 V=800.0 PL=0
MOVL C00794 V=800.0 PL=0
MOVL C00795 V=800.0 PL=0
MOVL C00796 V=800.0 PL=0
MOVL C00797 V=800.0 PL=0
MOVL C00798 V=800.0 PL=0
MOVL C00799 V=800.0 PL=0
MOVL C00800 V=800.0 PL=0
MOVL C00801 V=800.0 PL=0
MOVL C00802 V=800.0 PL=0
MOVL C00803 V=800.0 PL=0
MOVL C00804 V=800.0 PL=0
MOVL C00805 V=800.0 PL=0
MOVL C00806 V=800.0 PL=0
MOVL C00807 V=800.0 PL=0
MOVL C00808 V=800.0 PL=0
MOVL C00809 V=800.0 PL=0
MOVL C00810 V=800.0 PL=0
MOVL C00811 V=800.0 PL=0
MOVL C00812 V=800.0 PL=0
MOVL C00813 V=800.0 PL=0
MOVL C00814 V=800.0 PL=0
MOVL C00815 V=800.0 PL=0
MOVL C00816 V=800.0 PL=0
MOVL C00817 V=800.0 PL=0
MOVL C00818 V=800.0 PL=0
MOVL C00819 V=800.0 PL=0
MOVL C00820 V=800.0 PL=0
MOVL C00821 V=800.0 PL=0
MOVL C00822 V=800.0 PL=0
MOVL C00823 V=800.0 PL=0
MOVL C00824 V=800.0 PL=0
MOVL C00825 V=800.0 PL=0
MOVL C00826 V=800.0 PL=0
MOVL C00827 V=800.0 PL=0
MOVL C00828 V=800.0 PL=0
MOVL C00829 V=800.0 PL=0
MOVL C00830 V=800.0 PL=0
MOVL C00831 V=800.0 PL=0
MOVL C00832 V=800.0 PL=0
MOVL C00833 V=800.0 PL=0
MOVL C00834 V=800.0 PL=0
MOVL C00835 V=800.0 PL=0
MOVL C00836 V=800.0 PL=0
MOVL C00837 V=800.0 PL=0
MOVL C00838 V=800.0 PL=0
MOVL C00839 V=800.0 PL=0
MOVL C00840 V=800.0 PL=0
MOVL C00841 V=800.0 PL=0
MOVL C00842 V=800.0 PL=0
MOVL C00843 V=800.0 PL=0
MOVL C00844 V=800.0 PL=0
MOVL C00845 V=800.0 PL=0
MOVL C00846 V=800.0 PL=0
MOVL C00847 V=800.0 PL=0
MOVL C00848 V=800.0 PL=0
MOVL C00849 V=800.0 PL=0
MOVL C00850 V=800.0 PL=0
MOVL C00851 V=800.0 PL=0
MOVL C00852 V=800.0 PL=0
MOVL C00853 V=800.0 PL=0
MOVL C00854 V=800.0 PL=0
MOVL C00855 V=800.0 PL=0
MOVL C00856 V=800.0 PL=0
MOVL C00857 V=800.0 PL=0
MOVL C00858 V=800.0 PL=0
MOVL C00859 V=800.0 PL=0
MOVL C00860 V=800.0 PL=0
MOVL C00861 V=800.0 PL=0
MOVL C00862 V=800.0 PL=0
MOVL C00863 V=800.0 PL=0
MOVL C00864 V=800.0 PL=0
MOVL C00865 V=800.0 PL=0
MOVL C00866 V=800.0 PL=0
MOVL C00867 V=800.0 PL=0
MOVL C00868 V=800.0 PL=0
MOVL C00869 V=800.0 PL=0
MOVL C00870 V=800.0 PL=0
MOVL C00871 V=800.0 PL=0
MOVL C00872 V=800.0 PL=0
MOVL C00873 V=800.0 PL=0
MOVL C00874 V=800.0 PL=0
MOVL C00875 V=800.0 PL=0
MOVL C00876 V=800.0 PL=0
MOVL C00877 V=800.0 PL=0
MOVL C00878 V=800.0 PL=0
MOVL C00879 V=800.0 PL=0
MOVL C00880 V=800.0 PL=0
MOVL C00881 V=800.0 PL=0
MOVL C00882 V=800.0 PL=0
MOVL C00883 V=800.0 PL=0
MOVL C00884 V=800.0 PL=0
MOVL C00885 V=800.0 PL=0
MOVL C00886 V=800.0 PL=0
MOVL C00887 V=800.0 PL=0
MOVL C00888 V=800.0 PL=0
MOVL C00889 V=800.0 PL=0
MOVL C00890 V=800.0 PL=0
MOVL C00891 V=800.0 PL=0
MOVL C00892 V=800.0 PL=0
MOVL C00893 V=800.0 PL=0
MOVL C00894 V=800.0 PL=0
MOVL C00895 V=800.0 PL=0
MOVL C00896 V=800.0 PL=0
MOVL C00897 V=800.0 PL=0
MOVL C00898 V=800.0 PL=0
MOVL C00899 V=800.0 PL=0
MOVL C00900 V=800.0 PL=0
MOVL C00901 V=800.0 PL=0
MOVL C00902 V=800.0 PL=0
MOVL C00903 V=800.0 PL=0
MOVL C00904 V=800.0 PL=0
MOVL C00905 V=800.0 PL=0
MOVL C00906 V=800.0 PL=0
MOVL C00907 V=800.0 PL=0
MOVL C00908 V=800.0 PL=0
MOVL C00909 V=800.0 PL=0
MOVL C00910 V=800.0 PL=0
MOVL C00911 V=800.0 PL=0
MOVL C00912 V=800.0 PL=0
MOVL C00913 V=800.0 PL=0
MOVL C00914 V=800.0 PL=0
MOVL C00915 V=800.0 PL=0
MOVL C00916 V=800.0 PL=0
MOVL C00917 V=800.0 PL=0
MOVL C00918 V=800.0 PL=0
MOVL C00919 V=800.0 PL=0
MOVL C00920 V=800.0 PL=0
MOVL C00921 V=800.0 PL=0
MOVL C00922 V=800.0 PL=0
MOVL C00923 V=800.0 PL=0
MOVL C00924 V=800.0 PL=0
MOVL C00925 V=800.0 PL=0
MOVL C00926 V=800.0 PL=0
MOVL C00927 V=800.0 PL=0
MOVL C00928 V=800.0 PL=0
MOVL C00929 V=800.0 PL=0
MOVL C00930 V=800.0 PL=0
MOVL C00931 V=800.0 PL=0
MOVL C00932 V=800.0 PL=0
MOVL C00933 V=800.0 PL=0
MOVL C00934 V=800.0 PL=0
MOVL C00935 V=800.0 PL=0
MOVL C00936 V=800.0 PL=0
MOVL C00937 V=800.0 PL=0
MOVL C00938 V=800.0 PL=0
MOVL C00939 V=800.0 PL=0
MOVL C00940 V=800.0 PL=0
MOVL C00941 V=800.0 PL=0
MOVL C00942 V=800.0 PL=0
MOVL C00943 V=800.0 PL=0
MOVL C00944 V=800.0 PL=0
MOVL C00945 V=800.0 PL=0
MOVL C00946 V=800.0 PL=0
MOVL C00947 V=800.0 PL=0
MOVL C00948 V=800.0 PL=0
MOVL C00949 V=800.0 PL=0
MOVL C00950 V=800.0 PL=0
MOVL C00951 V=800.0 PL=0
MOVL C00952 V=800.0 PL=0
MOVL C00953 V=800.0 PL=0
MOVL C00954 V=800.0 PL=0
MOVL C00955 V=800.0 PL=0
MOVL C00956 V=800.0 PL=0
MOVL C00957 V=800.0 PL=0
MOVL C00958 V=800.0 PL=0
MOVL C00959 V=800.0 PL=0
MOVL C00960 V=800.0 PL=0
MOVL C00961 V=800.0 PL=0
MOVL C00962 V=800.0 PL=0
MOVL C00963 V=800.0 PL=0
MOVL C00964 V=800.0 PL=0
MOVL C00965 V=800.0 PL=0
MOVL C00966 V=800.0 PL=0
MOVL C00967 V=800.0 PL=0
MOVL C00968 V=800.0 PL=0
MOVL C00969 V=800.0 PL=0
MOVL C00970 V=800.0 PL=0
MOVL C00971 V=800.0 PL=0
MOVL C00972 V=800.0 PL=0
MOVL C00973 V=800.0 PL=0
MOVL C00974 V=800.0 PL=0
MOVL C00975 V=800.0 PL=0
MOVL C00976 V=800.0 PL=0
MOVL C00977 V=800.0 PL=0
MOVL C00978 V=800.0 PL=0
MOVL C00979 V=800.0 PL=0
MOVL C00980 V=800.0 PL=0
MOVL C00981 V=800.0 PL=0
MOVL C00982 V=800.0 PL=0
MOVL C00983 V=800.0 PL=0
MOVL C00984 V=800.0 PL=0
MOVL C00985 V=800.0 PL=0
MOVL C00986 V=800.0 PL=0
MOVL C00987 V=800.0 PL=0
MOVL C00988 V=800.0 PL=0
MOVL C00989 V=800.0 PL=0
MOVL C00990 V=800.0 PL=0
MOVL C00991 V=800.0 PL=0
MOVL C00992 V=800.0 PL=0
MOVL C00993 V=800.0 PL=0
MOVL C00994 V=800.0 PL=0
MOVL C00995 V=800.0 PL=0
MOVL C00996 V=800.0 PL=0
MOVL C00997 V=800.0 PL=0
MOVL C00998 V=800.0 PL=0
MOVL C00999 V=800.0 PL=0
MOVL C01000 V=800.0 PL=0
MOVL C01001 V=800.0 PL=0
MOVL C01002 V=800.0 PL=0
MOVL C01003 V=800.0 PL=0
MOVL C01004 V=800.0 PL=0
MOVL C01005 V=800.0 PL=0
MOVL C01006 V=800.0 PL=0
MOVL C01007 V=800.0 PL=0
MOVL C01008 V=800.0 PL=0
MOVL C01009 V=800.0 PL=0
MOVL C01010 V=800.0 PL=0
MOVL C01011 V=800.0 PL=0
MOVL C01012 V=800.0 PL=0
MOVL C01013 V=800.0 PL=0
MOVL C01014 V=800.0 PL=0
MOVL C01015 V=800.0 PL=0
MOVL C01016 V=800.0 PL=0
MOVL C01017 V=800.0 PL=0
MOVL C01018 V=800.0 PL=0
MOVL C01019 V=800.0 PL=0
MOVL C01020 V=800.0 PL=0
MOVL C01021 V=800.0 PL=0
MOVL C01022 V=800.0 PL=0
MOVL C01023 V=800.0 PL=0
MOVL C01024 V=800.0 PL=0
MOVL C01025 V=800.0 PL=0
MOVL C01026 V=800.0 PL=0
MOVL C01027 V=800.0 PL=0
MOVL C01028 V=800.0 PL=0
MOVL C01029 V=800.0 PL=0
MOVL C01030 V=800.0 PL=0
MOVL C01031 V=800.0 PL=0
MOVL C01032 V=800.0 PL=0
MOVL C01033 V=800.0 PL=0
MOVL C01034 V=800.0 PL=0
MOVL C01035 V=800.0 PL=0
MOVL C01036 V=800.0 PL=0
MOVL C01037 V=800.0 PL=0
MOVL C01038 V=800.0 PL=0
MOVL C01039 V=800.0 PL=0
MOVL C01040 V=800.0 PL=0
MOVL C01041 V=800.0 PL=0
MOVL C01042 V=800.0 PL=0
MOVL C01043 V=800.0 PL=0
MOVL C01044 V=800.0 PL=0
MOVL C01045 V=800.0 PL=0
MOVL C01046 V=800.0 PL=0
MOVL C01047 V=800.0 PL=0
MOVL C01048 V=800.0 PL=0
MOVL C01049 V=800.0 PL=0
MOVL C01050 V=800.0 PL=0
MOVL C01051 V=800.0 PL=0
MOVL C01052 V=800.0 PL=0
MOVL C01053 V=800.0 PL=0
MOVL C01054 V=800.0 PL=0
MOVL C01055 V=800.0 PL=0
MOVL C01056 V=800.0 PL=0
MOVL C01057 V=800.0 PL=0
MOVL C01058 V=800.0 PL=0
MOVL C01059 V=800.0 PL=0
MOVL C01060 V=800.0 PL=0
MOVL C01061 V=800.0 PL=0
MOVL C01062 V=800.0 PL=0
MOVL C01063 V=800.0 PL=0
MOVL C01064 V=800.0 PL=0
MOVL C01065 V=800.0 PL=0
MOVL C01066 V=800.0 PL=0
MOVL C01067 V=800.0 PL=0
MOVL C01068 V=800.0 PL=0
MOVL C01069 V=800.0 PL=0
MOVL C01070 V=800.0 PL=0
MOVL C01071 V=800.0 PL=0
MOVL C01072 V=800.0 PL=0
MOVL C01073 V=800.0 PL=0
MOVL C01074 V=800.0 PL=0
MOVL C01075 V=800.0 PL=0
MOVL C01076 V=800.0 PL=0
MOVL C01077 V=800.0 PL=0
MOVL C01078 V=800.0 PL=0
MOVL C01079 V=800.0 PL=0
MOVL C01080 V=800.0 PL=0
MOVL C01081 V=800.0 PL=0
MOVL C01082 V=800.0 PL=0
MOVL C01083 V=800.0 PL=0
MOVL C01084 V=800.0 PL=0
MOVL C01085 V=800.0 PL=0
MOVL C01086 V=800.0 PL=0
MOVL C01087 V=800.0 PL=0
MOVL C01088 V=800.0 PL=0
MOVL C01089 V=800.0 PL=0
MOVL C01090 V=800.0 PL=0
MOVL C01091 V=800.0 PL=0
MOVL C01092 V=800.0 PL=0
MOVL C01093 V=800.0 PL=0
MOVL C01094 V=800.0 PL=0
MOVL C01095 V=800.0 PL=0
MOVL C01096 V=800.0 PL=0
MOVL C01097 V=800.0 PL=0
MOVL C01098 V=800.0 PL=0
MOVL C01099 V=800.0 PL=0
MOVL C01100 V=800.0 PL=0
MOVL C01101 V=800.0 PL=0
MOVL C01102 V=800.0 PL=0
MOVL C01103 V=800.0 PL=0
MOVL C01104 V=800.0 PL=0
MOVL C01105 V=800.0 PL=0
MOVL C01106 V=800.0 PL=0
MOVL C01107 V=800.0 PL=0
MOVL C01108 V=800.0 PL=0
MOVL C01109 V=800.0 PL=0
MOVL C01110 V=800.0 PL=0
MOVL C01111 V=800.0 PL=0
MOVL C01112 V=800.0 PL=0
MOVL C01113 V=800.0 PL=0
MOVL C01114 V=800.0 PL=0
MOVL C01115 V=800.0 PL=0
MOVL C01116 V=800.0 PL=0
MOVL C01117 V=800.0 PL=0
MOVL C01118 V=800.0 PL=0
MOVL C01119 V=800.0 PL=0
MOVL C01120 V=800.0 PL=0
MOVL C01121 V=800.0 PL=0
MOVL C01122 V=800.0 PL=0
MOVL C01123 V=800.0 PL=0
MOVL C01124 V=800.0 PL=0
MOVL C01125 V=800.0 PL=0
MOVL C01126 V=800.0 PL=0
MOVL C01127 V=800.0 PL=0
MOVL C01128 V=800.0 PL=0
MOVL C01129 V=800.0 PL=0
MOVL C01130 V=800.0 PL=0
MOVL C01131 V=800.0 PL=0
MOVL C01132 V=800.0 PL=0
MOVL C01133 V=800.0 PL=0
MOVL C01134 V=800.0 PL=0
MOVL C01135 V=800.0 PL=0
MOVL C01136 V=800.0 PL=0
MOVL C01137 V=800.0 PL=0
MOVL C01138 V=800.0 PL=0
MOVL C01139 V=800.0 PL=0
MOVL C01140 V=800.0 PL=0
MOVL C01141 V=800.0 PL=0
MOVL C01142 V=800.0 PL=0
MOVL C01143 V=800.0 PL=0
MOVL C01144 V=800.0 PL=0
MOVL C01145 V=800.0 PL=0
MOVL C01146 V=800.0 PL=0
MOVL C01147 V=800.0 PL=0
MOVL C01148 V=800.0 PL=0
MOVL C01149 V=800.0 PL=0
MOVL C01150 V=800.0 PL=0
MOVL C01151 V=800.0 PL=0
MOVL C01152 V=800.0 PL=0
MOVL C01153 V=800.0 PL=0
MOVL C01154 V=800.0 PL=0
MOVL C01155 V=800.0 PL=0
MOVL C01156 V=800.0 PL=0
MOVL C01157 V=800.0 PL=0
MOVL C01158 V=800.0 PL=0
MOVL C01159 V=800.0 PL=0
MOVL C01160 V=800.0 PL=0
MOVL C01161 V=800.0 PL=0
MOVL C01162 V=800.0 PL=0
MOVL C01163 V=800.0 PL=0
MOVL C01164 V=800.0 PL=0
MOVL C01165 V=800.0 PL=0
MOVL C01166 V=800.0 PL=0
MOVL C01167 V=800.0 PL=0
MOVL C01168 V=800.0 PL=0
MOVL C01169 V=800.0 PL=0
MOVL C01170 V=800.0 PL=0
MOVL C01171 V=800.0 PL=0
MOVL C01172 V=800.0 PL=0
MOVL C01173 V=800.0 PL=0
MOVL C01174 V=800.0 PL=0
MOVL C01175 V=800.0 PL=0
MOVL C01176 V=800.0 PL=0
MOVL C01177 V=800.0 PL=0
MOVL C01178 V=800.0 PL=0
MOVL C01179 V=800.0 PL=0
MOVL C01180 V=800.0 PL=0
MOVL C01181 V=800.0 PL=0
MOVL C01182 V=800.0 PL=0
MOVL C01183 V=800.0 PL=0
MOVL C01184 V=800.0 PL=0
MOVL C01185 V=800.0 PL=0
MOVL C01186 V=800.0 PL=0
MOVL C01187 V=800.0 PL=0
MOVL C01188 V=800.0 PL=0
MOVL C01189 V=800.0 PL=0
MOVL C01190 V=800.0 PL=0
MOVL C01191 V=800.0 PL=0
MOVL C01192 V=800.0 PL=0
MOVL C01193 V=800.0 PL=0
MOVL C01194 V=800.0 PL=0
MOVL C01195 V=800.0 PL=0
MOVL C01196 V=800.0 PL=0
MOVL C01197 V=800.0 PL=0
MOVL C01198 V=800.0 PL=0
MOVL C01199 V=800.0 PL=0
MOVL C01200 V=800.0 PL=0
MOVL C01201 V=800.0 PL=0
MOVL C01202 V=800.0 PL=0
MOVL C01203 V=800.0 PL=0
MOVL C01204 V=800.0 PL=0
MOVL C01205 V=800.0 PL=0
MOVL C01206 V=800.0 PL=0
MOVL C01207 V=800.0 PL=0
MOVL C01208 V=800.0 PL=0
MOVL C01209 V=800.0 PL=0
MOVL C01210 V=800.0 PL=0
MOVL C01211 V=800.0 PL=0
MOVL C01212 V=800.0 PL=0
MOVL C01213 V=800.0 PL=0
MOVL C01214 V=800.0 PL=0
MOVL C01215 V=800.0 PL=0
MOVL C01216 V=800.0 PL=0
MOVL C01217 V=800.0 PL=0
MOVL C01218 V=800.0 PL=0
MOVL C01219 V=800.0 PL=0
MOVL C01220 V=800.0 PL=0
MOVL C01221 V=800.0 PL=0
MOVL C01222 V=800.0 PL=0
MOVL C01223 V=800.0 PL=0
MOVL C01224 V=800.0 PL=0
MOVL C01225 V=800.0 PL=0
MOVL C01226 V=800.0 PL=0
MOVL C01227 V=800.0 PL=0
MOVL C01228 V=800.0 PL=0
MOVL C01229 V=800.0 PL=0
MOVL C01230 V=800.0 PL=0
MOVL C01231 V=800.0 PL=0
MOVL C01232 V=800.0 PL=0
MOVL C01233 V=800.0 PL=0
MOVL C01234 V=800.0 PL=0
MOVL C01235 V=800.0 PL=0
MOVL C01236 V=800.0 PL=0
MOVL C01237 V=800.0 PL=0
MOVL C01238 V=800.0 PL=0
MOVL C01239 V=800.0 PL=0
MOVL C01240 V=800.0 PL=0
MOVL C01241 V=800.0 PL=0
MOVL C01242 V=800.0 PL=0
MOVL C01243 V=800.0 PL=0
MOVL C01244 V=800.0 PL=0
MOVL C01245 V=800.0 PL=0
MOVL C01246 V=800.0 PL=0
MOVL C01247 V=800.0 PL=0
MOVL C01248 V=800.0 PL=0
MOVL C01249 V=800.0 PL=0
MOVL C01250 V=800.0 PL=0
MOVL C01251 V=800.0 PL=0
MOVL C01252 V=800.0 PL=0
MOVL C01253 V=800.0 PL=0
MOVL C01254 V=800.0 PL=0
MOVL C01255 V=800.0 PL=0
MOVL C01256 V=800.0 PL=0
MOVL C01257 V=800.0 PL=0
MOVL C01258 V=800.0 PL=0
MOVL C01259 V=800.0 PL=0
MOVL C01260 V=800.0 PL=0
MOVL C01261 V=800.0 PL=0
MOVL C01262 V=800.0 PL=0
MOVL C01263 V=800.0 PL=0
MOVL C01264 V=800.0 PL=0
MOVL C01265 V=800.0 PL=0
MOVL C01266 V=800.0 PL=0
MOVL C01267 V=800.0 PL=0
MOVL C01268 V=800.0 PL=0
MOVL C01269 V=800.0 PL=0
MOVL C01270 V=800.0 PL=0
MOVL C01271 V=800.0 PL=0
MOVL C01272 V=800.0 PL=0
MOVL C01273 V=800.0 PL=0
MOVL C01274 V=800.0 PL=0
MOVL C01275 V=800.0 PL=0
MOVL C01276 V=800.0 PL=0
MOVL C01277 V=800.0 PL=0
MOVL C01278 V=800.0 PL=0
MOVL C01279 V=800.0 PL=0
MOVL C01280 V=800.0 PL=0
MOVL C01281 V=800.0 PL=0
MOVL C01282 V=800.0 PL=0
MOVL C01283 V=800.0 PL=0
MOVL C01284 V=800.0 PL=0
MOVL C01285 V=800.0 PL=0
MOVL C01286 V=800.0 PL=0
MOVL C01287 V=800.0 PL=0
MOVL C01288 V=800.0 PL=0
MOVL C01289 V=800.0 PL=0
MOVL C01290 V=800.0 PL=0
MOVL C01291 V=800.0 PL=0
MOVL C01292 V=800.0 PL=0
MOVL C01293 V=800.0 PL=0
MOVL C01294 V=800.0 PL=0
MOVL C01295 V=800.0 PL=0
MOVL C01296 V=800.0 PL=0
MOVL C01297 V=800.0 PL=0
MOVL C01298 V=800.0 PL=0
MOVL C01299 V=800.0 PL=0
MOVL C01300 V=800.0 PL=0
MOVL C01301 V=800.0 PL=0
MOVL C01302 V=800.0 PL=0
MOVL C01303 V=800.0 PL=0
MOVL C01304 V=800.0 PL=0
MOVL C01305 V=800.0 PL=0
MOVL C01306 V=800.0 PL=0
MOVL C01307 V=800.0 PL=0
MOVL C01308 V=800.0 PL=0
MOVL C01309 V=800.0 PL=0
MOVL C01310 V=800.0 PL=0
MOVL C01311 V=800.0 PL=0
MOVL C01312 V=800.0 PL=0
MOVL C01313 V=800.0 PL=0
MOVL C01314 V=800.0 PL=0
MOVL C01315 V=800.0 PL=0
MOVL C01316 V=800.0 PL=0
MOVL C01317 V=800.0 PL=0
MOVL C01318 V=800.0 PL=0
MOVL C01319 V=800.0 PL=0
MOVL C01320 V=800.0 PL=0
MOVL C01321 V=800.0 PL=0
MOVL C01322 V=800.0 PL=0
MOVL C01323 V=800.0 PL=0
MOVL C01324 V=800.0 PL=0
MOVL C01325 V=800.0 PL=0
MOVL C01326 V=800.0 PL=0
MOVL C01327 V=800.0 PL=0
MOVL C01328 V=800.0 PL=0
MOVL C01329 V=800.0 PL=0
MOVL C01330 V=800.0 PL=0
MOVL C01331 V=800.0 PL=0
MOVL C01332 V=800.0 PL=0
MOVL C01333 V=800.0 PL=0
MOVL C01334 V=800.0 PL=0
MOVL C01335 V=800.0 PL=0
MOVL C01336 V=800.0 PL=0
MOVL C01337 V=800.0 PL=0
MOVL C01338 V=800.0 PL=0
MOVL C01339 V=800.0 PL=0
MOVL C01340 V=800.0 PL=0
MOVL C01341 V=800.0 PL=0
MOVL C01342 V=800.0 PL=0
MOVL C01343 V=800.0 PL=0
MOVL C01344 V=800.0 PL=0
MOVL C01345 V=800.0 PL=0
MOVL C01346 V=800.0 PL=0
MOVL C01347 V=800.0 PL=0
MOVL C01348 V=800.0 PL=0
MOVL C01349 V=800.0 PL=0
MOVL C01350 V=800.0 PL=0
MOVL C01351 V=800.0 PL=0
MOVL C01352 V=800.0 PL=0
MOVL C01353 V=800.0 PL=0
MOVL C01354 V=800.0 PL=0
MOVL C01355 V=800.0 PL=0
MOVL C01356 V=800.0 PL=0
MOVL C01357 V=800.0 PL=0
MOVL C01358 V=800.0 PL=0
MOVL C01359 V=800.0 PL=0
MOVL C01360 V=800.0 PL=0
MOVL C01361 V=800.0 PL=0
MOVL C01362 V=800.0 PL=0
MOVL C01363 V=800.0 PL=0
MOVL C01364 V=800.0 PL=0
MOVL C01365 V=800.0 PL=0
MOVL C01366 V=800.0 PL=0
MOVL C01367 V=800.0 PL=0
MOVL C01368 V=800.0 PL=0
MOVL C01369 V=800.0 PL=0
MOVL C01370 V=800.0 PL=0
MOVL C01371 V=800.0 PL=0
MOVL C01372 V=800.0 PL=0
MOVL C01373 V=800.0 PL=0
MOVL C01374 V=800.0 PL=0
MOVL C01375 V=800.0 PL=0
MOVL C01376 V=800.0 PL=0
MOVL C01377 V=800.0 PL=0
MOVL C01378 V=800.0 PL=0
MOVL C01379 V=800.0 PL=0
MOVL C01380 V=800.0 PL=0
MOVL C01381 V=800.0 PL=0
MOVL C01382 V=800.0 PL=0
MOVL C01383 V=800.0 PL=0
MOVL C01384 V=800.0 PL=0
MOVL C01385 V=800.0 PL=0
MOVL C01386 V=800.0 PL=0
MOVL C01387 V=800.0 PL=0
MOVL C01388 V=800.0 PL=0
MOVL C01389 V=800.0 PL=0
MOVL C01390 V=800.0 PL=0
MOVL C01391 V=800.0 PL=0
MOVL C01392 V=800.0 PL=0
MOVL C01393 V=800.0 PL=0
MOVL C01394 V=800.0 PL=0
MOVL C01395 V=800.0 PL=0
MOVL C01396 V=800.0 PL=0
MOVL C01397 V=800.0 PL=0
MOVL C01398 V=800.0 PL=0
MOVL C01399 V=800.0 PL=0
MOVL C01400 V=800.0 PL=0
MOVL C01401 V=800.0 PL=0
MOVL C01402 V=800.0 PL=0
MOVL C01403 V=800.0 PL=0
MOVL C01404 V=800.0 PL=0
MOVL C01405 V=800.0 PL=0
MOVL C01406 V=800.0 PL=0
MOVL C01407 V=800.0 PL=0
MOVL C01408 V=800.0 PL=0
MOVL C01409 V=800.0 PL=0
MOVL C01410 V=800.0 PL=0
MOVL C01411 V=800.0 PL=0
MOVL C01412 V=800.0 PL=0
MOVL C01413 V=800.0 PL=0
MOVL C01414 V=800.0 PL=0
MOVL C01415 V=800.0 PL=0
MOVL C01416 V=800.0 PL=0
MOVL C01417 V=800.0 PL=0
MOVL C01418 V=800.0 PL=0
MOVL C01419 V=800.0 PL=0
MOVL C01420 V=800.0 PL=0
MOVL C01421 V=800.0 PL=0
MOVL C01422 V=800.0 PL=0
MOVL C01423 V=800.0 PL=0
MOVL C01424 V=800.0 PL=0
MOVL C01425 V=800.0 PL=0
MOVL C01426 V=800.0 PL=0
MOVL C01427 V=800.0 PL=0
MOVL C01428 V=800.0 PL=0
MOVL C01429 V=800.0 PL=0
MOVL C01430 V=800.0 PL=0
MOVL C01431 V=800.0 PL=0
MOVL C01432 V=800.0 PL=0
MOVL C01433 V=800.0 PL=0
MOVL C01434 V=800.0 PL=0
MOVL C01435 V=800.0 PL=0
MOVL C01436 V=800.0 PL=0
MOVL C01437 V=800.0 PL=0
MOVL C01438 V=800.0 PL=0
MOVL C01439 V=800.0 PL=0
MOVL C01440 V=800.0 PL=0
MOVL C01441 V=800.0 PL=0
MOVL C01442 V=800.0 PL=0
MOVL C01443 V=800.0 PL=0
MOVL C01444 V=800.0 PL=0
MOVL C01445 V=800.0 PL=0
MOVL C01446 V=800.0 PL=0
MOVL C01447 V=800.0 PL=0
MOVL C01448 V=800.0 PL=0
MOVL C01449 V=800.0 PL=0
MOVL C01450 V=800.0 PL=0
MOVL C01451 V=800.0 PL=0
MOVL C01452 V=800.0 PL=0
MOVL C01453 V=800.0 PL=0
MOVL C01454 V=800.0 PL=0
MOVL C01455 V=800.0 PL=0
MOVL C01456 V=800.0 PL=0
MOVL C01457 V=800.0 PL=0
MOVL C01458 V=800.0 PL=0
MOVL C01459 V=800.0 PL=0
MOVL C01460 V=800.0 PL=0
MOVL C01461 V=800.0 PL=0
MOVL C01462 V=800.0 PL=0
MOVL C01463 V=800.0 PL=0
MOVL C01464 V=800.0 PL=0
MOVL C01465 V=800.0 PL=0
MOVL C01466 V=800.0 PL=0
MOVL C01467 V=800.0 PL=0
MOVL C01468 V=800.0 PL=0
MOVL C01469 V=800.0 PL=0
MOVL C01470 V=800.0 PL=0
MOVL C01471 V=800.0 PL=0
MOVL C01472 V=800.0 PL=0
MOVL C01473 V=800.0 PL=0
MOVL C01474 V=800.0 PL=0
MOVL C01475 V=800.0 PL=0
MOVL C01476 V=800.0 PL=0
MOVL C01477 V=800.0 PL=0
MOVL C01478 V=800.0 PL=0
MOVL C01479 V=800.0 PL=0
MOVL C01480 V=800.0 PL=0
MOVL C01481 V=800.0 PL=0
MOVL C01482 V=800.0 PL=0
MOVL C01483 V=800.0 PL=0
MOVL C01484 V=800.0 PL=0
MOVL C01485 V=800.0 PL=0
MOVL C01486 V=800.0 PL=0
MOVL C01487 V=800.0 PL=0
MOVL C01488 V=800.0 PL=0
MOVL C01489 V=800.0 PL=0
MOVL C01490 V=800.0 PL=0
MOVL C01491 V=800.0 PL=0
MOVL C01492 V=800.0 PL=0
MOVL C01493 V=800.0 PL=0
MOVL C01494 V=800.0 PL=0
MOVL C01495 V=800.0 PL=0
MOVL C01496 V=800.0 PL=0
MOVL C01497 V=800.0 PL=0
MOVL C01498 V=800.0 PL=0
MOVL C01499 V=800.0 PL=0
MOVL C01500 V=800.0 PL=0
MOVL C01501 V=800.0 PL=0
MOVL C01502 V=800.0 PL=0
MOVL C01503 V=800.0 PL=0
MOVL C01504 V=800.0 PL=0
MOVL C01505 V=800.0 PL=0
MOVL C01506 V=800.0 PL=0
MOVL C01507 V=800.0 PL=0
MOVL C01508 V=800.0 PL=0
MOVL C01509 V=800.0 PL=0
MOVL C01510 V=800.0 PL=0
MOVL C01511 V=800.0 PL=0
MOVL C01512 V=800.0 PL=0
MOVL C01513 V=800.0 PL=0
MOVL C01514 V=800.0 PL=0
MOVL C01515 V=800.0 PL=0
MOVL C01516 V=800.0 PL=0
MOVL C01517 V=800.0 PL=0
MOVL C01518 V=800.0 PL=0
MOVL C01519 V=800.0 PL=0
MOVL C01520 V=800.0 PL=0
MOVL C01521 V=800.0 PL=0
MOVL C01522 V=800.0 PL=0
MOVL C01523 V=800.0 PL=0
MOVL C01524 V=800.0 PL=0
MOVL C01525 V=800.0 PL=0
MOVL C01526 V=800.0 PL=0
MOVL C01527 V=800.0 PL=0
MOVL C01528 V=800.0 PL=0
MOVL C01529 V=800.0 PL=0
MOVL C01530 V=800.0 PL=0
MOVL C01531 V=800.0 PL=0
MOVL C01532 V=800.0 PL=0
MOVL C01533 V=800.0 PL=0
MOVL C01534 V=800.0 PL=0
MOVL C01535 V=800.0 PL=0
MOVL C01536 V=800.0 PL=0
MOVL C01537 V=800.0 PL=0
MOVL C01538 V=800.0 PL=0
MOVL C01539 V=800.0 PL=0
MOVL C01540 V=800.0 PL=0
MOVL C01541 V=800.0 PL=0
MOVL C01542 V=800.0 PL=0
MOVL C01543 V=800.0 PL=0
MOVL C01544 V=800.0 PL=0
MOVL C01545 V=800.0 PL=0
MOVL C01546 V=800.0 PL=0
MOVL C01547 V=800.0 PL=0
MOVL C01548 V=800.0 PL=0
MOVL C01549 V=800.0 PL=0
MOVL C01550 V=800.0 PL=0
MOVL C01551 V=800.0 PL=0
MOVL C01552 V=800.0 PL=0
MOVL C01553 V=800.0 PL=0
MOVL C01554 V=800.0 PL=0
MOVL C01555 V=800.0 PL=0
MOVL C01556 V=800.0 PL=0
MOVL C01557 V=800.0 PL=0
MOVL C01558 V=800.0 PL=0
MOVL C01559 V=800.0 PL=0
MOVL C01560 V=800.0 PL=0
MOVL C01561 V=800.0 PL=0
MOVL C01562 V=800.0 PL=0
MOVL C01563 V=800.0 PL=0
MOVL C01564 V=800.0 PL=0
MOVL C01565 V=800.0 PL=0
MOVL C01566 V=800.0 PL=0
MOVL C01567 V=800.0 PL=0
MOVL C01568 V=800.0 PL=0
MOVL C01569 V=800.0 PL=0
MOVL C01570 V=800.0 PL=0
MOVL C01571 V=800.0 PL=0
MOVL C01572 V=800.0 PL=0
MOVL C01573 V=800.0 PL=0
MOVL C01574 V=800.0 PL=0
MOVL C01575 V=800.0 PL=0
MOVL C01576 V=800.0 PL=0
MOVL C01577 V=800.0 PL=0
MOVL C01578 V=800.0 PL=0
MOVL C01579 V=800.0 PL=0
MOVL C01580 V=800.0 PL=0
MOVL C01581 V=800.0 PL=0
MOVL C01582 V=800.0 PL=0
MOVL C01583 V=800.0 PL=0
MOVL C01584 V=800.0 PL=0
MOVL C01585 V=800.0 PL=0
MOVL C01586 V=800.0 PL=0
MOVL C01587 V=800.0 PL=0
MOVL C01588 V=800.0 PL=0
MOVL C01589 V=800.0 PL=0
MOVL C01590 V=800.0 PL=0
MOVL C01591 V=800.0 PL=0
MOVL C01592 V=800.0 PL=0
MOVL C01593 V=800.0 PL=0
MOVL C01594 V=800.0 PL=0
MOVL C01595 V=800.0 PL=0
MOVL C01596 V=800.0 PL=0
MOVL C01597 V=800.0 PL=0
MOVL C01598 V=800.0 PL=0
MOVL C01599 V=800.0 PL=0
MOVL C01600 V=800.0 PL=0
MOVL C01601 V=800.0 PL=0
MOVL C01602 V=800.0 PL=0
MOVL C01603 V=800.0 PL=0
MOVL C01604 V=800.0 PL=0
MOVL C01605 V=800.0 PL=0
MOVL C01606 V=800.0 PL=0
MOVL C01607 V=800.0 PL=0
MOVL C01608 V=800.0 PL=0
MOVL C01609 V=800.0 PL=0
MOVL C01610 V=800.0 PL=0
MOVL C01611 V=800.0 PL=0
MOVL C01612 V=800.0 PL=0
MOVL C01613 V=800.0 PL=0
MOVL C01614 V=800.0 PL=0
MOVL C01615 V=800.0 PL=0
MOVL C01616 V=800.0 PL=0
MOVL C01617 V=800.0 PL=0
MOVL C01618 V=800.0 PL=0
MOVL C01619 V=800.0 PL=0
MOVL C01620 V=800.0 PL=0
MOVL C01621 V=800.0 PL=0
MOVL C01622 V=800.0 PL=0
MOVL C01623 V=800.0 PL=0
MOVL C01624 V=800.0 PL=0
MOVL C01625 V=800.0 PL=0
MOVL C01626 V=800.0 PL=0
MOVL C01627 V=800.0 PL=0
MOVL C01628 V=800.0 PL=0
MOVL C01629 V=800.0 PL=0
MOVL C01630 V=800.0 PL=0
MOVL C01631 V=800.0 PL=0
MOVL C01632 V=800.0 PL=0
MOVL C01633 V=800.0 PL=0
MOVL C01634 V=800.0 PL=0
MOVL C01635 V=800.0 PL=0
MOVL C01636 V=800.0 PL=0
MOVL C01637 V=800.0 PL=0
MOVL C01638 V=800.0 PL=0
MOVL C01639 V=800.0 PL=0
MOVL C01640 V=800.0 PL=0
MOVL C01641 V=800.0 PL=0
MOVL C01642 V=800.0 PL=0
MOVL C01643 V=800.0 PL=0
MOVL C01644 V=800.0 PL=0
MOVL C01645 V=800.0 PL=0
MOVL C01646 V=800.0 PL=0
MOVL C01647 V=800.0 PL=0
MOVL C01648 V=800.0 PL=0
MOVL C01649 V=800.0 PL=0
MOVL C01650 V=800.0 PL=0
MOVL C01651 V=800.0 PL=0
MOVL C01652 V=800.0 PL=0
MOVL C01653 V=800.0 PL=0
MOVL C01654 V=800.0 PL=0
MOVL C01655 V=800.0 PL=0
MOVL C01656 V=800.0 PL=0
MOVL C01657 V=800.0 PL=0
MOVL C01658 V=800.0 PL=0
MOVL C01659 V=800.0 PL=0
MOVL C01660 V=800.0 PL=0
MOVL C01661 V=800.0 PL=0
MOVL C01662 V=800.0 PL=0
MOVL C01663 V=800.0 PL=0
MOVL C01664 V=800.0 PL=0
MOVL C01665 V=800.0 PL=0
MOVL C01666 V=800.0 PL=0
MOVL C01667 V=800.0 PL=0
MOVL C01668 V=800.0 PL=0
MOVL C01669 V=800.0 PL=0
MOVL C01670 V=800.0 PL=0
MOVL C01671 V=800.0 PL=0
MOVL C01672 V=800.0 PL=0
MOVL C01673 V=800.0 PL=0
MOVL C01674 V=800.0 PL=0
MOVL C01675 V=800.0 PL=0
MOVL C01676 V=800.0 PL=0
MOVL C01677 V=800.0 PL=0
MOVL C01678 V=800.0 PL=0
MOVL C01679 V=800.0 PL=0
MOVL C01680 V=800.0 PL=0
MOVL C01681 V=800.0 PL=0
MOVL C01682 V=800.0 PL=0
MOVL C01683 V=800.0 PL=0
MOVL C01684 V=800.0 PL=0
MOVL C01685 V=800.0 PL=0
MOVL C01686 V=800.0 PL=0
MOVL C01687 V=800.0 PL=0
MOVL C01688 V=800.0 PL=0
MOVL C01689 V=800.0 PL=0
MOVL C01690 V=800.0 PL=0
MOVL C01691 V=800.0 PL=0
MOVL C01692 V=800.0 PL=0
MOVL C01693 V=800.0 PL=0
MOVL C01694 V=800.0 PL=0
MOVL C01695 V=800.0 PL=0
MOVL C01696 V=800.0 PL=0
MOVL C01697 V=800.0 PL=0
MOVL C01698 V=800.0 PL=0
MOVL C01699 V=800.0 PL=0
MOVL C01700 V=800.0 PL=0
MOVL C01701 V=800.0 PL=0
MOVL C01702 V=800.0 PL=0
MOVL C01703 V=800.0 PL=0
MOVL C01704 V=800.0 PL=0
MOVL C01705 V=800.0 PL=0
MOVL C01706 V=800.0 PL=0
MOVL C01707 V=800.0 PL=0
MOVL C01708 V=800.0 PL=0
MOVL C01709 V=800.0 PL=0
MOVL C01710 V=800.0 PL=0
MOVL C01711 V=800.0 PL=0
MOVL C01712 V=800.0 PL=0
MOVL C01713 V=800.0 PL=0
MOVL C01714 V=800.0 PL=0
MOVL C01715 V=800.0 PL=0
MOVL C01716 V=800.0 PL=0
MOVL C01717 V=800.0 PL=0
MOVL C01718 V=800.0 PL=0
MOVL C01719 V=800.0 PL=0
MOVL C01720 V=800.0 PL=0
MOVL C01721 V=800.0 PL=0
MOVL C01722 V=800.0 PL=0
MOVL C01723 V=800.0 PL=0
MOVL C01724 V=800.0 PL=0
MOVL C01725 V=800.0 PL=0
MOVL C01726 V=800.0 PL=0
MOVL C01727 V=800.0 PL=0
MOVL C01728 V=800.0 PL=0
MOVL C01729 V=800.0 PL=0
MOVL C01730 V=800.0 PL=0
MOVL C01731 V=800.0 PL=0
MOVL C01732 V=800.0 PL=0
MOVL C01733 V=800.0 PL=0
MOVL C01734 V=800.0 PL=0
MOVL C01735 V=800.0 PL=0
MOVL C01736 V=800.0 PL=0
MOVL C01737 V=800.0 PL=0
MOVL C01738 V=800.0 PL=0
MOVL C01739 V=800.0 PL=0
MOVL C01740 V=800.0 PL=0
MOVL C01741 V=800.0 PL=0
MOVL C01742 V=800.0 PL=0
MOVL C01743 V=800.0 PL=0
MOVL C01744 V=800.0 PL=0
MOVL C01745 V=800.0 PL=0
MOVL C01746 V=800.0 PL=0
MOVL C01747 V=800.0 PL=0
MOVL C01748 V=800.0 PL=0
MOVL C01749 V=800.0 PL=0
MOVL C01750 V=800.0 PL=0
MOVL C01751 V=800.0 PL=0
MOVL C01752 V=800.0 PL=0
MOVL C01753 V=800.0 PL=0
MOVL C01754 V=800.0 PL=0
MOVL C01755 V=800.0 PL=0
MOVL C01756 V=800.0 PL=0
MOVL C01757 V=800.0 PL=0
MOVL C01758 V=800.0 PL=0
MOVL C01759 V=800.0 PL=0
MOVL C01760 V=800.0 PL=0
MOVL C01761 V=800.0 PL=0
MOVL C01762 V=800.0 PL=0
MOVL C01763 V=800.0 PL=0
MOVL C01764 V=800.0 PL=0
MOVL C01765 V=800.0 PL=0
MOVL C01766 V=800.0 PL=0
MOVL C01767 V=800.0 PL=0
MOVL C01768 V=800.0 PL=0
MOVL C01769 V=800.0 PL=0
MOVL C01770 V=800.0 PL=0
MOVL C01771 V=800.0 PL=0
MOVL C01772 V=800.0 PL=0
MOVL C01773 V=800.0 PL=0
MOVL C01774 V=800.0 PL=0
MOVL C01775 V=800.0 PL=0
MOVL C01776 V=800.0 PL=0
MOVL C01777 V=800.0 PL=0
MOVL C01778 V=800.0 PL=0
MOVL C01779 V=800.0 PL=0
MOVL C01780 V=800.0 PL=0
MOVL C01781 V=800.0 PL=0
MOVL C01782 V=800.0 PL=0
MOVL C01783 V=800.0 PL=0
MOVL C01784 V=800.0 PL=0
MOVL C01785 V=800.0 PL=0
MOVL C01786 V=800.0 PL=0
MOVL C01787 V=800.0 PL=0
MOVL C01788 V=800.0 PL=0
MOVL C01789 V=800.0 PL=0
MOVL C01790 V=800.0 PL=0
MOVL C01791 V=800.0 PL=0
MOVL C01792 V=800.0 PL=0
MOVL C01793 V=800.0 PL=0
MOVL C01794 V=800.0 PL=0
MOVL C01795 V=800.0 PL=0
MOVL C01796 V=800.0 PL=0
MOVL C01797 V=800.0 PL=0
MOVL C01798 V=800.0 PL=0
